(* Logix 5000 project; controller PBS_Perfusion vendor 1 type 14 code 217 rev 32.14; software revision 32.03; part 21 of 27 *)
(* tags used below, declared in another part *)
   ONS : DINT[3];
   REAL : DINT;

ADD_ON_INSTRUCTION P_VSD   (* revision 4.10 .01 Release, vendor Rockwell Automation, ExecutePrescan, ExecuteEnableInFalse *)
// Variable Speed Drive
// Revision note:
// See Instruction Help for a summary of changes, and see 4.10 Release Notes for details.
// Help:
// Copyright © Rockwell Automation, Inc.  All Rights Reserved.
// This Instruction controls and monitors a Variable-Speed (AC or DC) Drive
// and provides:
// *  Starting drive, stopping drive, jogging drive, setting speed reference and setting direction
// *  Monitoring of run feedback, display of actual drive status, including accel, decel, direction, speed
// *  Detection of Failure to Start, Failure to Stop, Drive Fault/Not Ready
// *  Monitoring of Permissive conditions to allow starting
// *  Monitoring of Interlock conditions to stop drive or prevent starting
// *  Simulation, providing feedback of a working drive while disabling outputs
// *  Monitoring of I/O communication faults
// *  Alarms for Fail to Start, Fail to Stop, Interlock Trip, Drive Fault/Not Ready, I/O Fault
// *  Operation in Hand, Maintenance, Override, Program and Operator Modes
// *  "Available" status for use by automation logic to know whether drive
//       can be controlled by other objects.
// *  Horn output for audible alert prior to starting motor.
// Command Sources are arbitrated by a P_CmdSrc Add-On Instruction instance.
// Command Sources: Operator, External, Program, Override, Maintenance, Out of
// Service, Hand.  Alarms are provided by P_Alarm Add-On Instruction instances.
// SUMMARY OF CHANGES FROM PREVIOUS VERSION (4.10.00)
// See 4.10 Release Notes for details.
// * Corrected handling of Start Horn on shed conditions.
// * Modified to lock out jog when jog time expires until jog commands are cleared
// * Modified to handle overlapping Horn and Jog times.
// SUMMARY OF CHANGES FROM PREVIOUS VERSION (4.00.02)
// See 4.10 Release Notes for details.
// * Changed availability to use input availability from interlocks.
// * Added Horn Status, Horn Inhibit.
// * Updated to P_CmdSrc V4.10.00.
// * Modified simulated run feedback to handle run at zero speed ref.
// * Added Cfg_HasMoreObj.
// SUMMARY OF CHANGES FROM PREVIOUS VERSION (4.00.00)
// See 4.00 Release Notes for details.
// * Corrected handling Allow Local when horn is enabled.
// SUMMARY OF CHANGES FROM PREVIOUS VERSION (3.5-11)
// See 4.00 Release Notes for details.
// * Changed "Mode" to "Command Source".
// * Added audible alert on commanded start.  Added unacked alarm count.
// * Changed Inf_ items to HMI_, and added Cfg_Area for security.
// * Changed Start / Stop / Fwd / Rev / Jog to StartFwd / StartRev /Stop / JogFwd / JogRev.
// * Deleted Cfg_PCmdClear; all Program Commands are now self-clearing.
// * All OCmds/MCmds and ORdys/MRdys are now Local Tags.
// * Added Sts_RdyAck and Sts_RdyReset for use by external objects.
// * Aligned ready bit naming with command bit names.
// * Added configurable decimal places for display on HMI.
// * Modifications to Output Datalink clamp limit restrictions / checking.
// * Changed delay / time configuration items to REAL seconds.
// * Updated Val_Sts to common enumeration across all motors and drives.
VAR_IN_OUT
   Ref_FaultCodeList : P_DescList[1]; {required}   // Tag containing List of Fault Codes (DINT) and their Descriptions (STRING)
END_VAR
VAR_INPUT
   Inp_SpeedFdbk : REAL; {visible}   // Speed Feedbak in Drive Units (typ. 0-32767 = 0 to max freq.)
   Inp_LastFaultCode : DINT; {visible}   // Most recent drive fault code (enumeration)
   Inp_Datalink : REAL;   // Auxiliary Signal (datalink) Input in Drive (raw) Units
   Inp_Ready : BOOL := 1; {visible}   // 1=Drive is ready to run
   Inp_Running : BOOL; {visible}   // 1=Drive is Running (active)
   Inp_CommandDir : BOOL := 1; {visible}   // 1=Drive is commanded Forward, 0=Drive is commanded Reverse
   Inp_ActualDir : BOOL := 1; {visible}   // 1=Drive is running Forward, 0=Drive is running Reverse
   Inp_Accelerating : BOOL; {visible}   // 1=Drive is accelerating
   Inp_Decelerating : BOOL; {visible}   // 1=Drive is decelerating
   Inp_Alarm : BOOL; {visible}   // 1=Drive has an Alarm Condition (see drive display or manual)
   Inp_Faulted : BOOL; {visible}   // 1=Drive has Faulted (see drive display or manual)
   Inp_AtSpeed : BOOL; {visible}   // 1=Drive is at commanded speed
   Inp_FwdPermOK : BOOL := 1; {visible}   // 1=Permissives OK, drive can start Forward
   Inp_FwdNBPermOK : BOOL := 1; {visible}   // 1=Non-Bypassable Permissives OK, drive can start Forward
   Inp_RevPermOK : BOOL := 1; {visible}   // 1=Permissives OK, drive can start Reverse
   Inp_RevNBPermOK : BOOL := 1; {visible}   // 1=Non-Bypassable Permissives OK, motor can start Reverse
   Inp_IntlkOK : BOOL := 1; {visible}   // 1=Interlocks OK, drive can start/run
   Inp_NBIntlkOK : BOOL := 1; {visible}   // 1=Non-Bypassable Interlocks OK, drive can start/run
   Inp_IntlkAvail : BOOL;   // 1 = Interlock Availibility OK
   Inp_IOFault : BOOL;   // Input Communication Status 0=OK, 1=fail
   Inp_Sim : BOOL;   // 1=Simulate working drive; 0=Start/Stop/ Monitor actual drive
   Inp_Hand : ALIAS FOR CmdSrc.Inp_Hand;
   Inp_Ovrd : ALIAS FOR CmdSrc.Inp_Ovrd;
   Inp_OvrdCmd : DINT;   // Override Command: 0=None, 1=Stop, 2=Start Fwd 3=Start Rev
   Inp_OvrdSpeed : REAL;   // Value to set Speed Reference in Override Mode (SpeedRef EU)
   Inp_OvrdOutDatalink : REAL;   // Value to set Output Datalink in Override Mode (OutDatalink EU)
   Inp_ExtInh : ALIAS FOR CmdSrc.Inp_ExtInh;
   Inp_HornInh : BOOL;   // 1 = Inhibit audible alert, 0 = Alllow audible alert
   Inp_Reset : BOOL;   // 1=Reset Shed Latches and Cleared Alarms
   Cfg_HasReverse : BOOL;   // 1=Drive can be run reverse, 0=Forward only
   Cfg_HasJog : BOOL;   // 1=Drive Jog Command enabled/visible, 0=Drive Jog Command not allowed
   Cfg_AllowLocal : BOOL;   // 1=Allow Local Start/Stop without alarm, 0=Start/Stop from HMI/prog only
   Cfg_HasRunFdbk : BOOL;   // 1=Drive provides feedback signal on Inp_Running when running
   Cfg_UseRunFdbk : BOOL;   // 1=Drive run feedback should be used for failure checking
   Cfg_HasSpeedFdbk : BOOL;   // 1=Drive provides speed feedback on Inp_SpeedFdbk
   Cfg_UseSpeedFdbk : BOOL := 1;   // 1=Drive speed determines running state, 0=state determined by drive Active input bit
   Cfg_HasInpDatalink : BOOL;   // 1=A signal is connected to Inp_Datalink
   Cfg_HasOutDatalink : BOOL;   // 1=A signal is connected to Out_Datalink
   Cfg_HasFwdPermObj : BOOL;   // 1=Tells HMI a P_Perm is connected to Inp_FwdPerm
   Cfg_HasRevPermObj : BOOL;   // 1=Tells HMI a P_Perm is connected to Inp_RevPerm
   Cfg_HasIntlkObj : BOOL;   // 1=Tells HMI a P_Intlk is connected to Inp_Intlk
   Cfg_HasResInhObj : BOOL;   // 1=Tells HMI a P_ResInh Restart Inhibit is connected
   Cfg_HasRunTimeObj : BOOL;   // 1=Tells HMI a P_RunTime is connected
   Cfg_HasMoreObj : BOOL;   // 1=Tells HMI an object with more info is available
   Cfg_SetTrack : BOOL := 1;   // 1=Settings track for unselected sources, 0=no tracking
   Cfg_SetTrackOvrdHand : BOOL;   // 1=Prog/Oper/Ext Settings track Override/Hand
   Cfg_OperStopPrio : BOOL;   // 1=OCmd_Stop any time, 0=OCmd_Stop only when Oper selected
   Cfg_ExtStopPrio : BOOL;   // 1=XCmd_Stop any time, 0=XCmd_Stop only when Ext selected
   Cfg_OCmdResets : BOOL;   // 1=New drive OCmd resets shed latches and cleared alarms, 0=OCmdReset req'd.
   Cfg_XCmdResets : BOOL;   // 1=New drive XCmd resets shed latches and cleared alarms, 0=XCmdReset req'd.
   Cfg_OvrdPermIntlk : BOOL;   // 1=Override ignores Bypassable Perm/ Intlk; 0=always use Perm/Intlk
   Cfg_ShedOnFailToStart : BOOL := 1;   // 1=Stop Motor and Alarm on Fail to Start; 0=Alarm only on Fail to Start
   Cfg_ShedOnIOFault : BOOL := 1;   // 1=Stop Motor and Alarm on I/O Fault; 0=Alarm only on I/O Fault
   Cfg_SimScaleEU : BOOL;   // 1=In simulation, scale Speed Ref EU to Speed Fdbk EU
   Cfg_SimScaleRaw : BOOL;   // 1=In simulation, scale Speed Ref EU to raw, then raw to Speed Fdbk EU
   Cfg_DecPlcs : DINT := 2;   // Number of decimal places for speed ref/fdbk display (0..6)
   Cfg_InpDLDecPlcs : DINT := 2;   // Number of decimal places for Input Datalink display (0..6)
   Cfg_OutDLDecPlcs : DINT := 2;   // Number of decimal places for Output Datalink display (0..6)
   Cfg_HasFailToStartAlm : ALIAS FOR FailToStart.Cfg_Exists;   // 1=Fail to Start Alarm exists and will be checked
   Cfg_HasFailToStopAlm : ALIAS FOR FailToStop.Cfg_Exists;   // 1=Fail to Stop Alarm exists and will be checked
   Cfg_HasIntlkTripAlm : ALIAS FOR IntlkTrip.Cfg_Exists;   // 1=Interlock Trip Alarm exists and will be checked
   Cfg_HasDriveFaultAlm : ALIAS FOR DriveFault.Cfg_Exists;   // 1=Drive Fault alarm exists and will be checked
   Cfg_HasIOFaultAlm : ALIAS FOR IOFault.Cfg_Exists;   // 1=I/O Fault Alarm exists and will be checked
   Cfg_FailToStartResetReqd : ALIAS FOR FailToStart.Cfg_ResetReqd;   // 1=Reset requied to clear Fail to Start Alarm
   Cfg_FailToStopResetReqd : ALIAS FOR FailToStop.Cfg_ResetReqd;   // 1=Reset required to clear Fail to Stop Alarm
   Cfg_IntlkTripResetReqd : ALIAS FOR IntlkTrip.Cfg_ResetReqd;   // 1=Reset required to clear Interlock Trip Alarm
   Cfg_DriveFaultResetReqd : ALIAS FOR DriveFault.Cfg_ResetReqd;   // 1=Reset required to clear Drive Fault Alarm
   Cfg_IOFaultResetReqd : ALIAS FOR IOFault.Cfg_ResetReqd;   // 1=Reset required to clear I/O Fault Alarm
   Cfg_FailToStartAckReqd : ALIAS FOR FailToStart.Cfg_AckReqd;   // 1=Acknowledge required for Fail to Start Alarm
   Cfg_FailToStopAckReqd : ALIAS FOR FailToStop.Cfg_AckReqd;   // 1=Acknowledge required for Fail to Stop Alarm
   Cfg_IntlkTripAckReqd : ALIAS FOR IntlkTrip.Cfg_AckReqd;   // 1=Acknowledge required for Interlock Trip Alarm
   Cfg_DriveFaultAckReqd : ALIAS FOR DriveFault.Cfg_AckReqd;   // 1=Acknowledge required for Drive Fault Alarm
   Cfg_IOFaultAckReqd : ALIAS FOR IOFault.Cfg_AckReqd;   // 1=Acknowledge required for I/O Fault Alarm
   Cfg_FailToStartSeverity : ALIAS FOR FailToStart.Cfg_Severity;   // Fail To Start Alarm Severity: 1..250=Low, 251..500=Medium, 501..750=High, 751..1000=Urgent
   Cfg_FailToStopSeverity : ALIAS FOR FailToStop.Cfg_Severity;   // Fail To Stop Alarm Severity: 1..250=Low, 251..500=Medium, 501..750=High, 751..1000=Urgent
   Cfg_IntlkTripSeverity : ALIAS FOR IntlkTrip.Cfg_Severity;   // Interlock Trip Alarm Severity: 1..250=Low, 251..500=Medium, 501..750=High, 751..1000=Urgent
   Cfg_DriveFaultSeverity : ALIAS FOR DriveFault.Cfg_Severity;   // Drive Fault Alarm Severity: 1..250=Low, 251..500=Medium, 501..750=High, 751..1000=Urgent
   Cfg_IOFaultSeverity : ALIAS FOR IOFault.Cfg_Severity;   // I/O Fault Alarm Severity: 1..250=Low, 251..500=Medium, 501..750=High, 751..1000=Urgent
   Cfg_MinSpdRef : REAL;   // Minimum Speed Reference in EU (for limiting)
   Cfg_MaxSpdRef : REAL := 60.0;   // Maximum Speed Reference in EU (for limiting)
   Cfg_SpeedRefRawMin : REAL;   // Speed Reference Minimum in Drive (raw) Units (for scaling)
   Cfg_SpeedRefRawMax : REAL := 32767.0;   // Speed Reference Maximum in Drive (raw) Units (for scaling)
   Cfg_SpeedRefEUMin : REAL;   // Speed Reference Minimum in Engineering Units (for scaling)
   Cfg_SpeedRefEUMax : REAL := 130.0;   // Speed Reference Maximum in Engineering Units (for scaling)
   Cfg_SpeedFdbkRawMin : REAL;   // Speed Feedback Minimum in Drive (raw) Units (for scaling)
   Cfg_SpeedFdbkRawMax : REAL := 32767.0;   // Speed Feedback Maximum in Drive (raw) Units (for scaling)
   Cfg_SpeedFdbkEUMin : REAL;   // Speed Feedback Minimum in Engineering Units (for scaling)
   Cfg_SpeedFdbkEUMax : REAL := 130.0;   // Speed Feedback Maximum in Engineering Units (for scaling)
   Cfg_InpDatalinkRawMin : REAL;   // Input Datalink Minimum in Drive (raw) Units (for scaling)
   Cfg_InpDatalinkRawMax : REAL := 4095.0;   // Input Datalink Maximum in Drive (raw) Units (for scaling)
   Cfg_InpDatalinkEUMin : REAL;   // Input Datalink Minimum in Engineering Units (for scaling)
   Cfg_InpDatalinkEUMax : REAL := 409.5;   // Input Datalink Maximum in Engineering Units (for scaling)
   Cfg_OutDatalinkMin : REAL;   // Minimum Output Datalink in EU (for limiting)
   Cfg_OutDatalinkMax : REAL := 100.0;   // Maximum Output Datalink in EU (for limiting)
   Cfg_OutDatalinkRawMin : REAL;   // Output Datalink Minimum in Drive (raw) Units (for scaling)
   Cfg_OutDatalinkRawMax : REAL := 4095.0;   // Output Datalink Maximum in Drive (raw) Units (for scaling)
   Cfg_OutDatalinkEUMin : REAL;   // Output Datalink Minimum in Engineering Units (for scaling)
   Cfg_OutDatalinkEUMax : REAL := 409.5;   // Output Datalink Maximum in Engineering Units (for scaling)
   Cfg_StartHornT : REAL;   // Time to sound audible on commanded start (sec) (0=disabled)
   Cfg_SimRampT : REAL := 10.0;   // Time to ramp speed fdbk when in Simulation (sec)
   Cfg_FailToStartT : REAL := 15.0;   // Time after Start to get Run Feedback before Fault (sec)
   Cfg_FailToStopT : REAL := 15.0;   // Time after Stop to drop Run Feedback before Fault (sec)
   Cfg_ResetPulseT : REAL := 2.0;   // Time to pulse Out_Reset to clear drive fault
   Cfg_MaxJogT : REAL;   // Maximum jog time (sec, 0=unlimited)
   Cfg_OperKeep : SINT;   // Oper keeps control in Prog / Ext: .0=Reference, .1=Start/Stop/Fwd/ Rev, .3=OutDatalink
   Cfg_ProgKeep : SINT;   // Prog keeps control in Oper / Ext: .0=Reference, .1=Start/Stop/Fwd/ Rev, .3=OutDatalink
   Cfg_ExtKeep : SINT;   // Ext keeps control in Prog / Oper: .0=Reference, .1=Start/Stop/Fwd/ Rev, .3=OutDatalink
   PSet_SpeedRef : REAL;   // Program Setting of Speed Reference (EU)
   PSet_OutDatalink : REAL;   // Program Setting of Output Datalink (EU)
   PSet_Owner : DINT;   // Program Owner Request ID (non-zero) or Release (zero)
   XSet_SpeedRef : REAL;   // External Setting of Speed Reference (EU)
   XSet_OutDatalink : REAL;   // External Setting of Output Datalink (EU)
   PCmd_StartFwd : BOOL;   // Program Command to Start Drive Forward
   PCmd_StartRev : BOOL;   // Program Command to Start Drive Reverse
   PCmd_Stop : BOOL;   // Program Command to Stop Drive
   PCmd_Prog : ALIAS FOR CmdSrc.PCmd_Prog;
   PCmd_Oper : ALIAS FOR CmdSrc.PCmd_Oper;
   PCmd_Lock : ALIAS FOR CmdSrc.PCmd_Lock;
   PCmd_Unlock : ALIAS FOR CmdSrc.PCmd_Unlock;
   PCmd_Normal : ALIAS FOR CmdSrc.PCmd_Normal;
   PCmd_Reset : BOOL;   // Program Command to Reset drive fault and all Alarms requiring Reset
   PCmd_FailToStartAck : ALIAS FOR FailToStart.PCmd_Ack;   // Program Command to Acknowledge Fail to Start Alarm
   PCmd_FailToStartSuppress : ALIAS FOR FailToStart.PCmd_Suppress;   // Program Command to Suppress Fail to Start Alarm
   PCmd_FailToStartUnsuppress : ALIAS FOR FailToStart.PCmd_Unsuppress;   // Program Command to Unsuppress Fail to Start Alarm
   PCmd_FailToStartUnshelve : ALIAS FOR FailToStart.PCmd_Unshelve;   // Program Command to Unshelve Fail to Start Alarm
   PCmd_FailToStopAck : ALIAS FOR FailToStop.PCmd_Ack;   // Program Command to Acknowledge Fail to Stop Alarm
   PCmd_FailToStopSuppress : ALIAS FOR FailToStop.PCmd_Suppress;   // Program Command to Suppress Fail to Stop Alarm
   PCmd_FailToStopUnsuppress : ALIAS FOR FailToStop.PCmd_Unsuppress;   // Program Command to Unsuppress Fail to Stop Alarm
   PCmd_FailToStopUnshelve : ALIAS FOR FailToStop.PCmd_Unshelve;   // Program Command to Unshelve Fail to Stop Alarm
   PCmd_IntlkTripAck : ALIAS FOR IntlkTrip.PCmd_Ack;   // Program Command to Acknowledge Interlock Trip Alarm
   PCmd_IntlkTripSuppress : ALIAS FOR IntlkTrip.PCmd_Suppress;   // Program Command to Suppress Interlock Trip Alarm
   PCmd_IntlkTripUnsuppress : ALIAS FOR IntlkTrip.PCmd_Unsuppress;   // Program Command to Unsuppress Interlock Trip Alarm
   PCmd_IntlkTripUnshelve : ALIAS FOR IntlkTrip.PCmd_Unshelve;   // Program Command to Unshelve Interlock Trip Alarm
   PCmd_DriveFaultAck : ALIAS FOR DriveFault.PCmd_Ack;   // Program Command to Acknowledge Drive Fault Alarm
   PCmd_DriveFaultSuppress : ALIAS FOR DriveFault.PCmd_Suppress;   // Program Command to Suppress Drive Fault Alarm
   PCmd_DriveFaultUnsuppress : ALIAS FOR DriveFault.PCmd_Unsuppress;   // Program Command to Unsuppress Drive Fault Alarm
   PCmd_DriveFaultUnshelve : ALIAS FOR DriveFault.PCmd_Unshelve;   // Program Command to Unshelve Drive Fault Alarm
   PCmd_IOFaultAck : ALIAS FOR IOFault.PCmd_Ack;   // Program Command to Acknowledge I/O Fault Alarm
   PCmd_IOFaultSuppress : ALIAS FOR IOFault.PCmd_Suppress;   // Program Command to Suppress I/O Fault Alarm
   PCmd_IOFaultUnsuppress : ALIAS FOR IOFault.PCmd_Unsuppress;   // Program Command to Unsuppress I/O Fault Alarm
   PCmd_IOFaultUnshelve : ALIAS FOR IOFault.PCmd_Unshelve;   // Program Command to Unshelve I/O Fault Alarm
   MCmd_Rel : ALIAS FOR CmdSrc.MCmd_Rel;
   OCmd_Unlock : ALIAS FOR CmdSrc.OCmd_Unlock;
   XCmd_StartFwd : BOOL;   // External Command to Start Drive Forward
   XCmd_StartRev : BOOL;   // External Command to Start Drive Reverse
   XCmd_Stop : BOOL;   // External Command to Stop Drive
   XCmd_JogFwd : BOOL;   // External Command to Jog Drive Forward
   XCmd_JogRev : BOOL;   // External Command to Jog Drive Reverse
   XCmd_Acq : ALIAS FOR CmdSrc.XCmd_Acq;
   XCmd_Rel : ALIAS FOR CmdSrc.XCmd_Rel;
   XCmd_Reset : BOOL;   // Ext Cmd to clear shed latches and cleared alarms
END_VAR
VAR_OUTPUT
   Out_SpeedRef : REAL; {access Read Only, visible}   // Drive Speed Reference in Drive Units (typ. 0-32767 = 0 to max freq.)
   Out_Datalink : REAL; {access Read Only, visible}   // Auxiliary Signal (datalink) Output in Drive (raw) Units
   Out_Run : BOOL; {access Read Only}   // 1=Start/Run Drive, 0=Stop Drive (for held starter type)
   Out_Stop : BOOL; {access Read Only, visible}   // 1=Stop Drive, 0=drive left in current state
   Out_Start : BOOL; {access Read Only, visible}   // 1=Start Drive, 0=drive left in current state
   Out_Jog : BOOL; {access Read Only, visible}   // 1=Jog drive at Jog Speed, -->0=stop jogging
   Out_ClearFault : BOOL; {access Read Only, visible}   // 1=Attempt to clear Drive Fault
   Out_Fwd : BOOL; {access Read Only, visible}   // 1=Set drive direction to Forward
   Out_Rev : BOOL; {access Read Only, visible}   // 1=Set drive direction to Reverse
   Out_Horn : BOOL; {access Read Only, visible}   // 1=Sound audible prior to commanded motor start
   Val_SpeedRef : REAL; {access Read Only, visible}   // Speed Reference (target) to drive
   Val_SpeedFdbk : REAL; {access Read Only, visible}   // Speed Feedback (actual) from drive
   Val_InpDatalink : REAL; {access Read Only, visible}   // Input Datalink value from drive
   Val_OutDatalink : REAL; {access Read Only, visible}   // Output Datalink value to drive
   Val_SpeedRefEUMin : REAL; {access Read Only}   // Minimum of Speed Reference = MIN (Cfg_SpeedFdbkEUMin, Cfg_SpeedFdbkEUMax)
   Val_SpeedRefEUMax : REAL := 130.0; {access Read Only}   // Maximum of Speed Reference = MAX (Cfg_SpeedFdbkEUMin, Cfg_SpeedFdbkEUMax)
   Val_SpeedFdbkEUMin : REAL; {access Read Only}   // Minimum of Speed Feedback = MIN (Cfg_SpeedFdbkEUMin, Cfg_SpeedFdbkEUMax)
   Val_SpeedFdbkEUMax : REAL := 130.0; {access Read Only}   // Maximum of Speed Feedback = MAX (Cfg_SpeedFdbkEUMin, Cfg_SpeedFdbkEUMax)
   Val_LastFaultCode : DINT; {access Read Only}   // Most recent drive fault code (enumeration)
   SrcQ_IO : DINT; {access Read Only}   // Source and Quality of primary I/O (enumeration)
   SrcQ : DINT; {access Read Only}   // Source and Quality of primary Val/Sts (enumeration)
   Val_Cmd : DINT; {access Read Only}   // Device Command 0=None, 1=Stop, 2=StartFwd 3=StartRev 4=JogFwd 5=JogRev
   Val_Fdbk : DINT; {access Read Only}   // Device Feedback 0=Stopped, 1=Running Fwd 2=Running Rev 3=Accelerating 4=Decelerating
   Val_Sts : DINT; {access Read Only}   // Device Sts: 0=? 1=Stopped 2=RunFwd 3=RunRev 4=RunSlow 5=StartFwd 6=StartRev 7=StartSlow 8=JogFwd 9=JogRev 10=Stopping
   Val_Fault : DINT; {access Read Only, visible}   // Device Fault Status 0=None, 16=Fail to Start, 17 = Fail to Stop, 18=Drive Fault, 32=I/O Fault, 34=Config Error
   Val_NotifyAll : DINT; {access Read Only}   // Highest Alarm prio and ack status this object + channel (enum)
   Val_UnackAlmC : DINT; {access Read Only}   // Count of Unacknowledged Alarms
   Val_Owner : DINT; {access Read Only}   // Current Object Owner ID (0=not owned)
   Sts_Stopped : BOOL; {access Read Only, visible}   // 1=Drive requested to stop and is confirmed stopped
   Sts_StartingFwd : BOOL; {access Read Only, visible}   // 1=Drive requested to run forward and awaiting run feedback
   Sts_StartingRev : BOOL; {access Read Only, visible}   // 1=Drive requested to run reverse and awaiting run feedback
   Sts_RunningFwd : BOOL; {access Read Only, visible}   // 1=Drive requested to run and is confirmed running forward
   Sts_RunningRev : BOOL; {access Read Only, visible}   // 1=Drive requested to run and is confirmed running reverse
   Sts_StoppingFwd : BOOL; {access Read Only, visible}   // 1=Drive running forward requested to stop and awaiting stopped feedback
   Sts_StoppingRev : BOOL; {access Read Only, visible}   // 1=Drive running reverse requested to stop and awaiting stopped feedback
   Sts_JoggingFwd : BOOL; {access Read Only, visible}   // 1=Drive requested to Jog Forward
   Sts_JoggingRev : BOOL; {access Read Only, visible}   // 1=Drive requested to Jog Reverse
   Sts_Horn : BOOL; {access Read Only}   // 1=Motor Horn Active
   Sts_CommandDir : BOOL; {access Read Only}   // 1=Drive commanded to Forward, 0=Reverse
   Sts_ActualDir : BOOL; {access Read Only, visible}   // 1=Drive Actual direction is Forward, 0=Reverse
   Sts_Accel : BOOL; {access Read Only}   // 1=Drive is Accelerating
   Sts_Decel : BOOL; {access Read Only}   // 1=Drive is Decelerating
   Sts_NotReady : BOOL; {access Read Only}   // 1=Drive is Not Ready (cannot be started) Check alarms, stops, faults
   Sts_Alarm : BOOL; {access Read Only, visible}   // 1=Drive has an Alarm (see drive display or manual)
   Sts_AtSpeed : BOOL; {access Read Only, visible}   // 1=Drive is running at reference speed
   Sts_SpeedLimited : BOOL; {access Read Only, visible}   // 1=Speed Reference Setting exceeds configured Max/Min limit
   Sts_Available : BOOL; {access Read Only, visible}   // 1=Drive available for control by automation (Prog)
   Sts_Bypass : BOOL; {access Read Only}   // 1=Bypassable Interlocks and Permissives are Bypassed
   Sts_BypActive : BOOL; {access Read Only}   // 1=Bypassing Active (Bypassed or Maintenance)
   Sts_NotRdy : BOOL; {access Read Only}   // 1=Device Not Ready, see detail bits for reason
   Nrdy_CfgErr : BOOL; {access Read Only}   // 1=Device Not Ready: Configuration Error
   Nrdy_DriveNR : BOOL; {access Read Only}   // 1=Device Note Ready: Drive Not Ready
   Nrdy_Fail : BOOL; {access Read Only}   // 1=Device Not Ready: Device Failure (Shed Requires Reset)
   Nrdy_Intlk : BOOL; {access Read Only, visible}   // 1=Device Not Ready: Interlock Not OK
   Nrdy_IOFault : BOOL; {access Read Only}   // 1=Device Not Ready: I/O Fault (Shed Requires Reset)
   Nrdy_OoS : BOOL; {access Read Only}   // 1=Device Not Ready: Device is Out of Service
   Nrdy_Perm : BOOL; {access Read Only}   // 1=Device Not Ready: Permissive Not OK
   Nrdy_PrioStop : BOOL; {access Read Only}   // 1=Device Not Ready: Oper/Ext Priority Stop Requires Reset
   Nrdy_Trip : BOOL; {access Read Only}   // 1=Device not Ready: Deivce Tripped (Drive Fault)
   Sts_MaintByp : BOOL; {access Read Only}   // 1=A Maintenance Bypass is Active, display icon
   Sts_AlmInh : BOOL; {access Read Only}   // 1=An Alarm is Shelved, Disabled or Suppressed, display icon
   Sts_Err : BOOL; {access Read Only, visible}   // 1=Error in Config: see detail bits for reason
   Err_Timer : BOOL; {access Read Only}   // 1=Error in Config: Invalid Check or Reset Pulse Time (use 0 to 2147483)
   Err_Sim : BOOL; {access Read Only}   // 1=Error in Config: simulation timer preset: use 0 to 2147483)
   Err_Alarm : BOOL; {access Read Only}   // 1=Error in Config: Alarm Min On Time, Shelf Time, Severity
   Err_FdbkRaw : BOOL; {access Read Only}   // 1=Erron in Config: Speed Fdbk Raw Min = Max
   Err_FdbkEU : BOOL; {access Read Only}   // 1=Error in Config: Speed Fdbk EU Min = Max
   Err_RefLim : BOOL; {access Read Only}   // 1=Error in Config: Speed Ref Limit Min > Max
   Err_RefEU : BOOL; {access Read Only}   // 1=Error in Config: Speed Ref EU Min = Max
   Err_RefRaw : BOOL; {access Read Only}   // 1=Error in Config: Speed Ref Raw Min = Max
   Err_InpDLRaw : BOOL; {access Read Only}   // 1=Error in Config: Input Datalink Raw Min = Max
   Err_InpDLEU : BOOL; {access Read Only}   // 1=Error in Config: Input Datalink EU Min = Max
   Err_OutDLLim : BOOL; {access Read Only}   // 1=Error in Config: Output Datalink Limits Min > Max
   Err_OutDLEU : BOOL; {access Read Only}   // 1=Error in Config: Output Datalink EU Min = Max
   Err_OutDLRaw : BOOL; {access Read Only}   // 1=Error in Config: Output Datalink Raw Min = Max
   Sts_Hand : ALIAS FOR CmdSrc.Sts_Hand; {access Read Only, visible}
   Sts_OoS : ALIAS FOR CmdSrc.Sts_OoS; {access Read Only, visible}
   Sts_Maint : ALIAS FOR CmdSrc.Sts_Maint; {access Read Only, visible}
   Sts_Ovrd : ALIAS FOR CmdSrc.Sts_Ovrd; {access Read Only, visible}
   Sts_Ext : ALIAS FOR CmdSrc.Sts_Ext; {access Read Only, visible}
   Sts_Prog : ALIAS FOR CmdSrc.Sts_Prog; {access Read Only, visible}
   Sts_ProgLocked : ALIAS FOR CmdSrc.Sts_ProgLocked; {access Read Only}
   Sts_Oper : ALIAS FOR CmdSrc.Sts_Oper; {access Read Only, visible}
   Sts_OperLocked : ALIAS FOR CmdSrc.Sts_OperLocked; {access Read Only}
   Sts_Normal : ALIAS FOR CmdSrc.Sts_Normal; {access Read Only}
   Sts_ExtReqInh : ALIAS FOR CmdSrc.Sts_ExtReqInh; {access Read Only}
   Sts_ProgReqInh : ALIAS FOR CmdSrc.Sts_ProgReqInh; {access Read Only}
   Sts_MAcqRcvd : ALIAS FOR CmdSrc.Sts_MAcqRcvd; {access Read Only}
   Sts_RdyReset : ALIAS FOR ORdy_Reset; {access Read Only}   // 1=A latched alarm or shed condition is ready to be reset
   Sts_RdyAck : BOOL; {access Read Only}   // 1=An alarm is ready to be acknowledged
   Sts_FailToStart : ALIAS FOR FailToStart.Inp;   // 1=Drive Failed to Start (One-Shot)
   Alm_FailToStart : ALIAS FOR FailToStart.Alm;   // 1=Drive Fail to Start Alarm
   Ack_FailToStart : ALIAS FOR FailToStart.Ack;   // 1=Fail to Start Alarm has been acknowledged
   Sts_FailToStartDisabled : ALIAS FOR FailToStart.Disabled;   // 1=Fail to Start Alarm has been Disabled by Maintenance
   Sts_FailToStartShelved : ALIAS FOR FailToStart.Shelved;   // 1=Fail to Start Alarm has been Shelved by Operator
   Sts_FailToStartSuppressed : ALIAS FOR FailToStart.Suppressed;   // 1=Fail to Start Alarm has been Suppressed by Program
   Sts_FailToStop : ALIAS FOR FailToStop.Inp;   // 1=Drive Failed to Stop
   Alm_FailToStop : ALIAS FOR FailToStop.Alm;   // 1=Drive Fail to Stop Alarm
   Ack_FailToStop : ALIAS FOR FailToStop.Ack;   // 1=Fail to Stop Alarm has been acknowledged
   Sts_FailToStopDisabled : ALIAS FOR FailToStop.Disabled;   // 1=Fail to Stop Alarm has been Disabled by Maintenance
   Sts_FailToStopShelved : ALIAS FOR FailToStop.Shelved;   // 1=Fail to Stop Alarm has been Shelved by Operator
   Sts_FailToStopSuppressed : ALIAS FOR FailToStop.Suppressed;   // 1=Fail to Stop Alarm has been Suppressed by Program
   Sts_IntlkTrip : ALIAS FOR IntlkTrip.Inp;   // 1=Drive was stopped by an Interlock NOT OK (One-Shot)
   Alm_IntlkTrip : ALIAS FOR IntlkTrip.Alm;   // 1=Alarm: Drive stopped by an Interlock NOT OK
   Ack_IntlkTrip : ALIAS FOR IntlkTrip.Ack;   // 1=Interlock Trip Alarm has been acknowledged
   Sts_IntlkTripDisabled : ALIAS FOR IntlkTrip.Disabled;   // 1=Interlock Trip Alarm has been Disabled by Maintenance
   Sts_IntlkTripShelved : ALIAS FOR IntlkTrip.Shelved;   // 1=Interlock Trip Alarm has been Shelved by Operator
   Sts_IntlkTripSuppressed : ALIAS FOR IntlkTrip.Suppressed;   // 1=Interlock Trip Alarm has been Suppressed by Program
   Sts_DriveFault : ALIAS FOR DriveFault.Inp;   // 1=Drive Fault (see drive display or manual)
   Alm_DriveFault : ALIAS FOR DriveFault.Alm;   // 1=Alarm: Drive Fault (see drive display or manual)
   Ack_DriveFault : ALIAS FOR DriveFault.Ack;   // 1=Drive Fault Alarm has been acknowledged
   Sts_DriveFaultDisabled : ALIAS FOR DriveFault.Disabled;   // 1=Drive Fault Alarm has been Disabled by Maintenance
   Sts_DriveFaultShelved : ALIAS FOR DriveFault.Shelved;   // 1=Drive Fault Alarm has been Shelved by Operator
   Sts_DriveFaultSuppressed : ALIAS FOR DriveFault.Suppressed;   // 1=Drive Fault Alarm has been Suppressed by Program
   Sts_IOFault : ALIAS FOR IOFault.Inp;   // I/O Comm Fault Status (0=OK, 1=Bad)
   Alm_IOFault : ALIAS FOR IOFault.Alm;   // 1=I/O Fault Alarm
   Ack_IOFault : ALIAS FOR IOFault.Ack;   // 1=I/O Fault Alarm has been acknowledged
   Sts_IOFaultDisabled : ALIAS FOR IOFault.Disabled;   // 1=I/O Fault Alarm has been Disabled by Maintenance
   Sts_IOFaultShelved : ALIAS FOR IOFault.Shelved;   // 1=I/O Fault Alarm has been Shelved by Operator
   Sts_IOFaultSuppressed : ALIAS FOR IOFault.Suppressed;   // 1=I/O Fault Alarm has been Suppressed by Program
   MRdy_Rel : ALIAS FOR CmdSrc.MRdy_Rel; {access Read Only}
   ORdy_Unlock : ALIAS FOR CmdSrc.ORdy_Unlock; {access Read Only}
   P_VSD : BOOL;   // Unique Parameter Name for auto - discovery
END_VAR
VAR
   CmdSrc : P_CmdSrc := (Cfg_HasOper := 1, Cfg_HasOperLocked := 1, Cfg_HasProg := 1, Cfg_HasProgLocked := 1, Cfg_HasMaint := 1, Cfg_HasMOoS := 1, Cfg_OvrdOverLock := 1, Sts_bSrc := 1);   // Drive Mode Selection
   IOFault : P_Alarm := (Cfg_AckReqd := 1, Cfg_AllowShelve := 1, Cfg_AllowDisable := 1, Cfg_Severity := 1000, Cfg_AlmMinOnT := 5, PCfg_AllowExist := 1, Ack := 1);   // I/O Fault Alarm
   IntlkTrip : P_Alarm := (Cfg_AckReqd := 1, Cfg_AllowShelve := 1, Cfg_AllowDisable := 1, Cfg_Severity := 500, Cfg_AlmMinOnT := 5, PCfg_AllowExist := 1, Ack := 1);   // Interlock Trip Alarm
   FailToStop : P_Alarm := (Cfg_AckReqd := 1, Cfg_AllowShelve := 1, Cfg_AllowDisable := 1, Cfg_Severity := 1000, Cfg_AlmMinOnT := 5, PCfg_AllowExist := 1, Ack := 1);   // Drive Failed to Stop Alarm
   FailToStart : P_Alarm := (Cfg_AckReqd := 1, Cfg_AllowShelve := 1, Cfg_AllowDisable := 1, Cfg_Severity := 1000, Cfg_AlmMinOnT := 5, PCfg_AllowExist := 1, Ack := 1);   // Drive Failed to Start Alarm
   Cfg_Tag : STRING_20 := 'P_VSD';   // Tagname for display on HMI
   Cfg_Label : STRING_20 := 'Motor Speed Control';   // Label for graphic symbol displayed on HMI
   Cfg_Desc : STRING_40 := 'Variable Speed Drive';   // Description for display on HMI
   Wrk_Run : BOOL; {access None}   // 1=Drive should be "running", 0=should be "stopped"
   Wrk_StartRetrigT : TIMER; {access None}   // Time to pulse start output on start command retrigger (Maint)
   Wrk_StopRetrigT : TIMER; {access None}   // Time to pulse stop output on stop command retrigger (Maint)
   Wrk_RunFdbk : BOOL; {access None}   // Run Feedback based on mode, simulation, etc. 1=running
   Wrk_Notify : DINT; {access None}   // Buffer for building Val_Notify
   Wrk_Bypass : BOOL; {access None}   // Internal Bypassable Permissives and Interlocks are Bypassed flag
   DriveFault : P_Alarm := (Cfg_AckReqd := 1, Cfg_AllowShelve := 1, Cfg_AllowDisable := 1, Cfg_Severity := 1000, Cfg_AlmMinOnT := 5, PCfg_AllowExist := 1, Ack := 1);   // Drive Faulted Alarm
   Cfg_SpeedRefEU : STRING_8 := 'Hz';   // Speed Reference Engineering Units for display on HMI
   Wrk_SpeedRef : REAL; {access None}   // Working copy of Speed Reference (for limiting)
   Wrk_Rev : BOOL; {access None}   // Working (internal) Direction 1=Reverse 0=Forward (default)
   Wrk_Jog : BOOL; {access None}   // 1=Jog Drive, 0=Drive not jogging
   Wrk_ResetT : TIMER; {access None}   // Reset Output Pulse Timer
   Wrk_ResetONS : BOOL; {access None}   // One-Shot to fire Reset Timer to ensure min. output ON time.
   Cfg_SpeedFdbkEU : STRING_8 := 'Hz';   // Speed Feedback Engineering Units for display on HMI
   Cfg_OutDatalinkLabel : STRING_20;   // Datalink Output Label displayed on faceplate
   Cfg_InpDatalinkLabel : STRING_20;   // Datalink Input Label displayed on faceplate
   Cfg_OutDatalinkEU : STRING_8;   // Datalink Output Engineering Units for display on HMI
   Cfg_InpDatalinkEU : STRING_8;   // Datalink Input Engineering Units for display on HMI
   Wrk_OutDatalink : REAL; {access None}   // Selected Output Datalink setting
   Cfg_RevText : STRING_16 := 'Reverse';   // Name for Reverse Direction, e.g., "Down", "Reverse"
   Cfg_FwdText : STRING_16 := 'Forward';   // Name for Forward Direction, e.g., "Up", "Forward"
   Wrk_StopT : TIMER; {access Read Only}   // Stop Check Timer (for Fail to Stop)
   Wrk_StartT : TIMER; {access Read Only}   // Start Check Timer (for Fail to Start)
   HMI_Tab : SINT;   // Tab to display (FTView ME)
   Wrk_Cmd : DINT; {access None}   // Buffer for building Val_Cmd
   Wrk_Sts : DINT; {access None}   // Buffer for building Val_Sts
   Wrk_Fault : DINT; {access None}   // Buffer for building Val_Fault
   Wrk_Retrigger : BOOL; {access None}   // Maint Start issued while running or Stop while stopped
   Wrk_Step : REAL; {access None}   // Amount to change simulated Speed Fdbk this scan (ramp)
   Wrk_ScanTime : REAL; {access None}   // Seconds since previous scan
   Wrk_ScanT : TIMER := (PRE := 2147483647); {access None}   // Scan Timer (milliseconds, always runs)
   Wrk_SimFdbkTgt : REAL; {access None}   // Speed Ref converted to Speed Fdbk units for simulation: target speed fdbk
   HMI_Type : STRING_16 := 'P_VSD'; {access Read Only}   // Type identifier for HMI navigation
   Wrk_JogT : TIMER; {access Read Only}   // Jog Timer
   Wrk_FaultDescFSC : CONTROL := (LEN := 1); {access None}   // FSC control for Fault Code List search
   Val_FaultDesc : STRING_40; {access Read Only}   // Description of Drive Fault (given LastFaultCode)
   Wrk_OperKeep3ONS : BOOL; {access None}   // Oper Keep bit 3 one-shot store
   Wrk_OperKeep1ONS : BOOL; {access None}   // Oper Keep bit 1 one-shot store
   Wrk_OperKeep0ONS : BOOL; {access None}   // Oper Keep bit 0 one-shot store
   Wrk_ProgKeep3ONS : BOOL; {access None}   // Prog Keep bit 3 one-shot store
   Wrk_ProgKeep1ONS : BOOL; {access None}   // Prog Keep bit 1 one-shot store
   Wrk_ProgKeep0ONS : BOOL; {access None}   // Prog Keep bit 0 one-shot store
   HMI_Lib : STRING_12 := 'RA-BAS'; {access Read Only}   // Display Library for Faceplate call-up
   Wrk_SimScaleEUONS : BOOL; {access None}   // Cfg_SimScaleEU became true this scan
   Wrk_SimScaleRawONS : BOOL; {access None}   // Cfg_SimScaleRaw became true this scan
   Wrk_SrcQ : DINT; {access None}   // Register for building Source / Quality enumeration
   Val_Notify : DINT; {access Read Only}   // Current Alarm Level and Acknowledgement (enumeration)
   Wrk_NotRdyONS : BOOL; {access None}   // Assert Stop on One-Shot of Sts_NotRdy
   Wrk_NotRdy : BOOL; {access None}   // Device Not Ready conditions excluding shed latches
   Wrk_StartInhT : TIMER; {access None}   // Local Start Inhibit Timer
   Wrk_StopInhT : TIMER; {access None}   // Local Stop Inhibit Timer
   Wrk_NoLongerSim : BOOL; {access None}   // Switched from Simulated to Real Drive this scan
   Wrk_Hand : BOOL; {access None}   // Perform Hand Mode alignment with actual device state
   Cfg_Area : STRING_Area := 'area01';   // Process Area for security
   Wrk_UnackAlmC : DINT; {access None}   // Buffer for building Val_UnackAlmC
   Wrk_StartHornT : TIMER; {access None}   // Timer for audible alert or start
   Wrk_StartHorn : BOOL; {access None}   // 1=Sound audible prior to commanded motor start
   Wrk_RevPermOK : BOOL; {access None}   // Reverse Permissives and NB Permissive OK
   Wrk_FwdPermOK : BOOL; {access None}   // Forward Permissives and NB Permissive OK
   OCmd_ResetAckAll : BOOL;   // Oper Cmd to reset shed latches and cleared alarms, plus Acknowledge alarms
   OCmd_Reset : BOOL;   // Oper Cmd to clear shed latches and cleared alarms
   OCmd_JogRev : BOOL;   // Operator Command to Jog Drive Reverse (not cleared by instruction!)
   OCmd_JogFwd : BOOL;   // Operator Command to Jog Drive Forward (not cleared by instruction!)
   OCmd_Stop : BOOL;   // Operator Command to Stop Drive
   OCmd_StartRev : BOOL;   // Operator Command to Start Drive Reverse
   OCmd_StartFwd : BOOL;   // Operator Command to Start Drive Forward
   MCmd_Check : BOOL;   // Maintenance Command to Check (not bypass) all Interlocks and Permissives
   MCmd_Bypass : BOOL;   // Maintenance Command to Bypass all Bypassable Interlocks and Permissives
   OSet_OutDatalink : REAL;   // Operator Setting of Output Datalink (EU)
   OSet_SpeedRef : REAL;   // Operator Setting of Speed Reference (EU)
   ORdy_ResetAckAll : BOOL; {access Read Only}   // 1=Ready for OCmd_ResetAckAll (enables HMI button)
   ORdy_Reset : BOOL; {access Read Only}   // 1=Ready for OCmd_Reset (enables HMI button)
   ORdy_JogRev : BOOL; {access Read Only}   // 1=Ready for OCmd_JogRev (enabled HMI button)
   ORdy_JogFwd : BOOL; {access Read Only}   // 1=Ready for OCmd_JogFwd (enables HMI button)
   ORdy_Stop : BOOL; {access Read Only}   // 1=Ready for OCmd_Stop (enables HMI button)
   ORdy_StartRev : BOOL; {access Read Only}   // 1=Ready for OCmd_StartRev (enables HMI button)
   ORdy_StartFwd : BOOL; {access Read Only}   // 1=Ready for OCmd_StartFwd (enables HMI button)
   ORdy_OSet : BOOL; {access Read Only}   // 1=Ready for OSets (other than Speed Ref) (enables data entry fields)
   ORdy_SpeedRef : BOOL; {access Read Only}   // 1=Ready for OSet_SpeedRef (enables data entry field)
   MRdy_Check : BOOL; {access Read Only}   // 1=Ready for MCmd_Check (enables HMI button)
   MRdy_Bypass : BOOL; {access Read Only}   // 1=Ready for MCmd_Bypass (enables HMI button)
   Wrk_ExtKeep3ONS : BOOL; {access None}   // Ext Keep bit 3 one-shot store
   Wrk_ExtKeep1ONS : BOOL; {access None}   // Ext Keep bit 1 one-shot store
   Wrk_ExtKeep0ONS : BOOL; {access None}   // Ext Keep bit 0 one-shot store
   Wrk_ExtHas3 : BOOL; {access None}   // External has Output Datalink
   Wrk_ExtHas1 : BOOL; {access None}   // External has Commands
   Wrk_ExtHas0 : BOOL; {access None}   // External has Speed Reference
   Wrk_ProgHas3 : BOOL; {access None}   // Program has Output Datalink
   Wrk_ProgHas1 : BOOL; {access None}   // Program has Commands
   Wrk_ProgHas0 : BOOL; {access None}   // Program has Speed Reference
   Wrk_OperHas3 : BOOL; {access None}   // Operator has Output Datalink
   Wrk_OperHas1 : BOOL; {access None}   // Operator has Commands
   Wrk_OperHas0 : BOOL; {access None}   // Operator has Speed Reference
END_VAR

ROUTINE EnableInFalse   (* ladder *)
// Out of Service is asserted; Outputs OFF; Run Status shown but Alarms inhibited
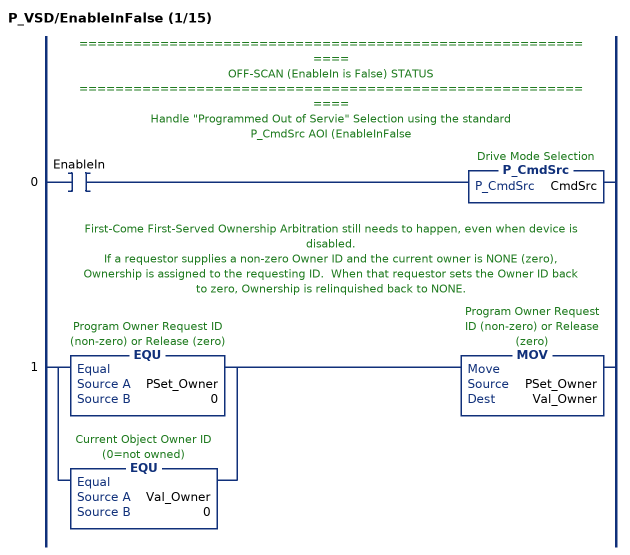
   // ============================================================
   // OFF-SCAN (EnableIn is False) STATUS
   // ============================================================
   // Handle "Programmed Out of Servie" Selection using the standard
   // P_CmdSrc AOI (EnableInFalse
   0: XIC(EnableIn)P_CmdSrc(CmdSrc);
   // First-Come First-Served Ownership Arbitration still needs to happen, even when device is disabled.
   // If a requestor supplies a non-zero Owner ID and the current owner is NONE (zero),
   // Ownership is assigned to the requesting ID.  When that requestor sets the Owner ID back
   // to zero, Ownership is relinquished back to NONE.
   1: [EQU(PSet_Owner,0) ,EQU(Val_Owner,0) ]MOV(PSet_Owner,Val_Owner);
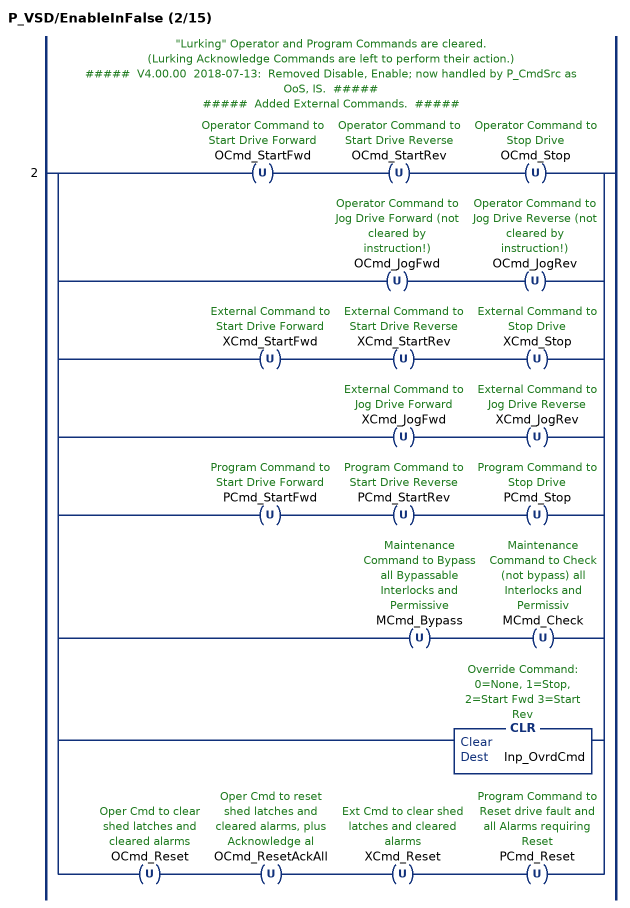
   // "Lurking" Operator and Program Commands are cleared.
   // (Lurking Acknowledge Commands are left to perform their action.)
   // #####  V4.00.00  2018-07-13:  Removed Disable, Enable; now handled by P_CmdSrc as OoS, IS.  #####
   // #####  Added External Commands.  #####
   2: [OTU(OCmd_StartFwd) OTU(OCmd_StartRev) OTU(OCmd_Stop) ,OTU(OCmd_JogFwd) OTU(OCmd_JogRev) ,OTU(XCmd_StartFwd) OTU(XCmd_StartRev) OTU(XCmd_Stop) ,OTU(XCmd_JogFwd) OTU(XCmd_JogRev) ,OTU(PCmd_StartFwd) OTU(PCmd_StartRev) OTU(PCmd_Stop) ,OTU(MCmd_Bypass) OTU(MCmd_Check) ,CLR(Inp_OvrdCmd) ,OTU(OCmd_Reset) OTU(OCmd_ResetAckAll) OTU(XCmd_Reset) OTU(PCmd_Reset) ];
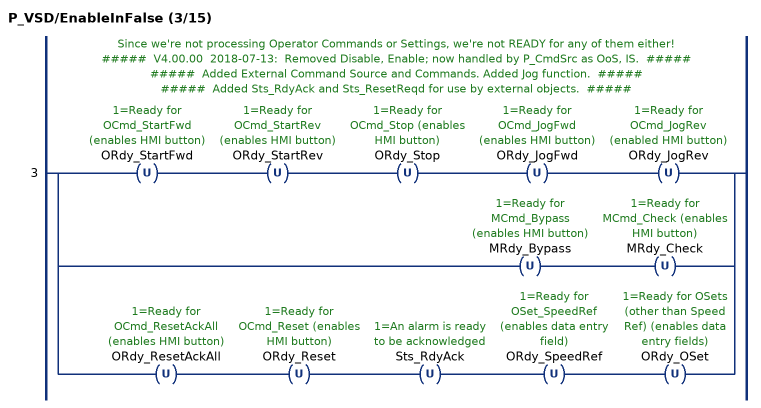
   // Since we're not processing Operator Commands or Settings, we're not READY for any of them either!
   // #####  V4.00.00  2018-07-13:  Removed Disable, Enable; now handled by P_CmdSrc as OoS, IS.  #####
   // #####  Added External Command Source and Commands. Added Jog function.  #####
   // #####  Added Sts_RdyAck and Sts_ResetReqd for use by external objects.  #####
   3: [OTU(ORdy_StartFwd) OTU(ORdy_StartRev) OTU(ORdy_Stop) OTU(ORdy_JogFwd) OTU(ORdy_JogRev) ,OTU(MRdy_Bypass) OTU(MRdy_Check) ,OTU(ORdy_ResetAckAll) OTU(ORdy_Reset) OTU(Sts_RdyAck) OTU(ORdy_SpeedRef) OTU(ORdy_OSet) ];
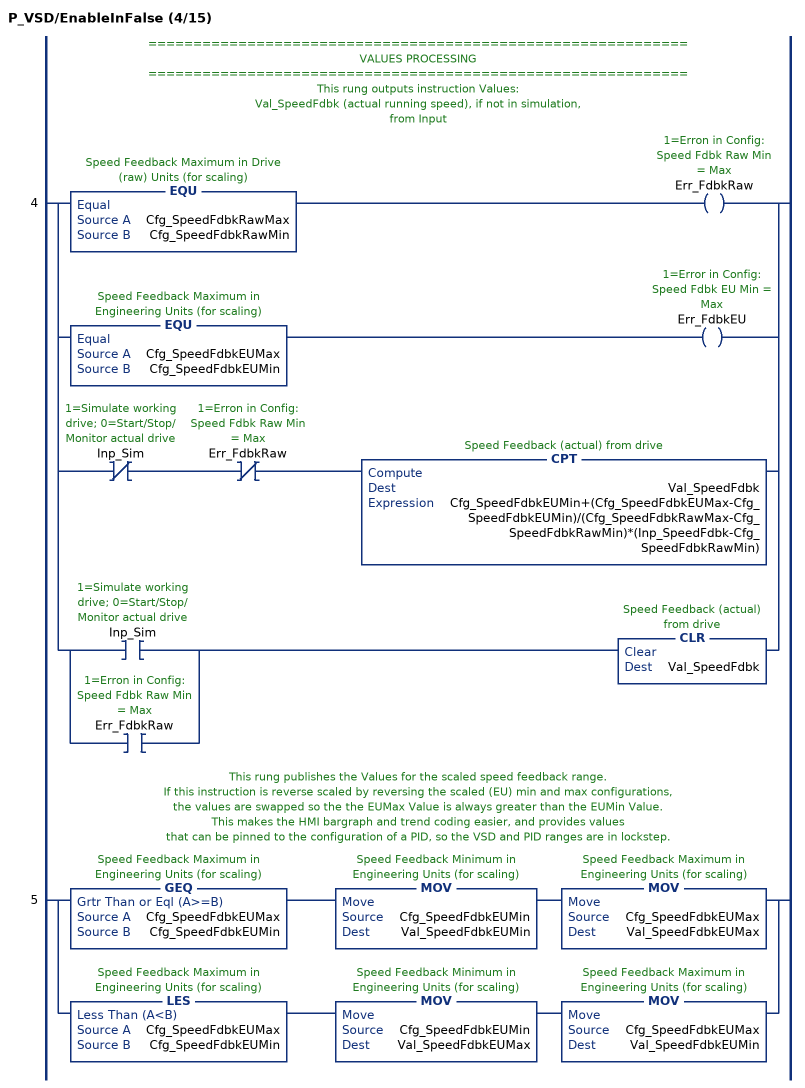
   // ============================================================
   // VALUES PROCESSING
   // ============================================================
   // This rung outputs instruction Values:
   // Val_SpeedFdbk (actual running speed), if not in simulation,
   // from Input
   4: [[EQU(Cfg_SpeedFdbkRawMax,Cfg_SpeedFdbkRawMin) OTE(Err_FdbkRaw) ,EQU(Cfg_SpeedFdbkEUMax,Cfg_SpeedFdbkEUMin) OTE(Err_FdbkEU) ] ,XIO(Inp_Sim) XIO(Err_FdbkRaw) CPT(Val_SpeedFdbk,Cfg_SpeedFdbkEUMin+(Cfg_SpeedFdbkEUMax-Cfg_SpeedFdbkEUMin)/(Cfg_SpeedFdbkRawMax-Cfg_SpeedFdbkRawMin)*(Inp_SpeedFdbk-Cfg_SpeedFdbkRawMin)) ,[XIC(Inp_Sim) ,XIC(Err_FdbkRaw) ] CLR(Val_SpeedFdbk) ];
   // This rung publishes the Values for the scaled speed feedback range.
   // If this instruction is reverse scaled by reversing the scaled (EU) min and max configurations,
   // the values are swapped so the the EUMax Value is always greater than the EUMin Value.
   // This makes the HMI bargraph and trend coding easier, and provides values
   // that can be pinned to the configuration of a PID, so the VSD and PID ranges are in lockstep.
   5: [GEQ(Cfg_SpeedFdbkEUMax,Cfg_SpeedFdbkEUMin) MOV(Cfg_SpeedFdbkEUMin,Val_SpeedFdbkEUMin) MOV(Cfg_SpeedFdbkEUMax,Val_SpeedFdbkEUMax) ,LES(Cfg_SpeedFdbkEUMax,Cfg_SpeedFdbkEUMin) MOV(Cfg_SpeedFdbkEUMin,Val_SpeedFdbkEUMax) MOV(Cfg_SpeedFdbkEUMax,Val_SpeedFdbkEUMin) ];
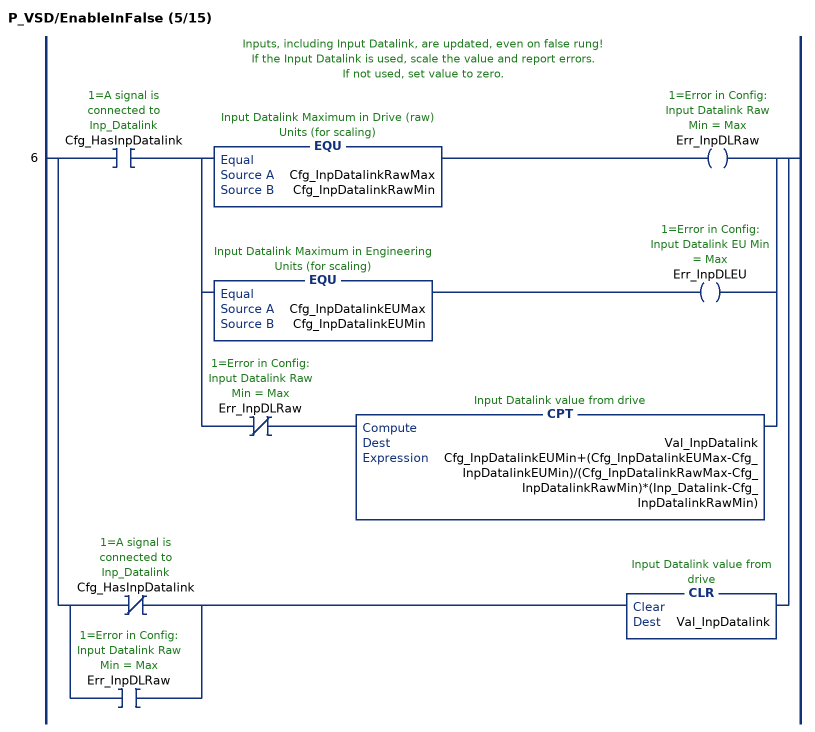
   // Inputs, including Input Datalink, are updated, even on false rung!
   // If the Input Datalink is used, scale the value and report errors.
   // If not used, set value to zero.
   6: [XIC(Cfg_HasInpDatalink) [[EQU(Cfg_InpDatalinkRawMax,Cfg_InpDatalinkRawMin) OTE(Err_InpDLRaw) ,EQU(Cfg_InpDatalinkEUMax,Cfg_InpDatalinkEUMin) OTE(Err_InpDLEU) ] ,XIO(Err_InpDLRaw) CPT(Val_InpDatalink,Cfg_InpDatalinkEUMin+(Cfg_InpDatalinkEUMax-Cfg_InpDatalinkEUMin)/(Cfg_InpDatalinkRawMax-Cfg_InpDatalinkRawMin)*(Inp_Datalink-Cfg_InpDatalinkRawMin)) ] ,[XIO(Cfg_HasInpDatalink) ,XIC(Err_InpDLRaw) ] CLR(Val_InpDatalink) ];
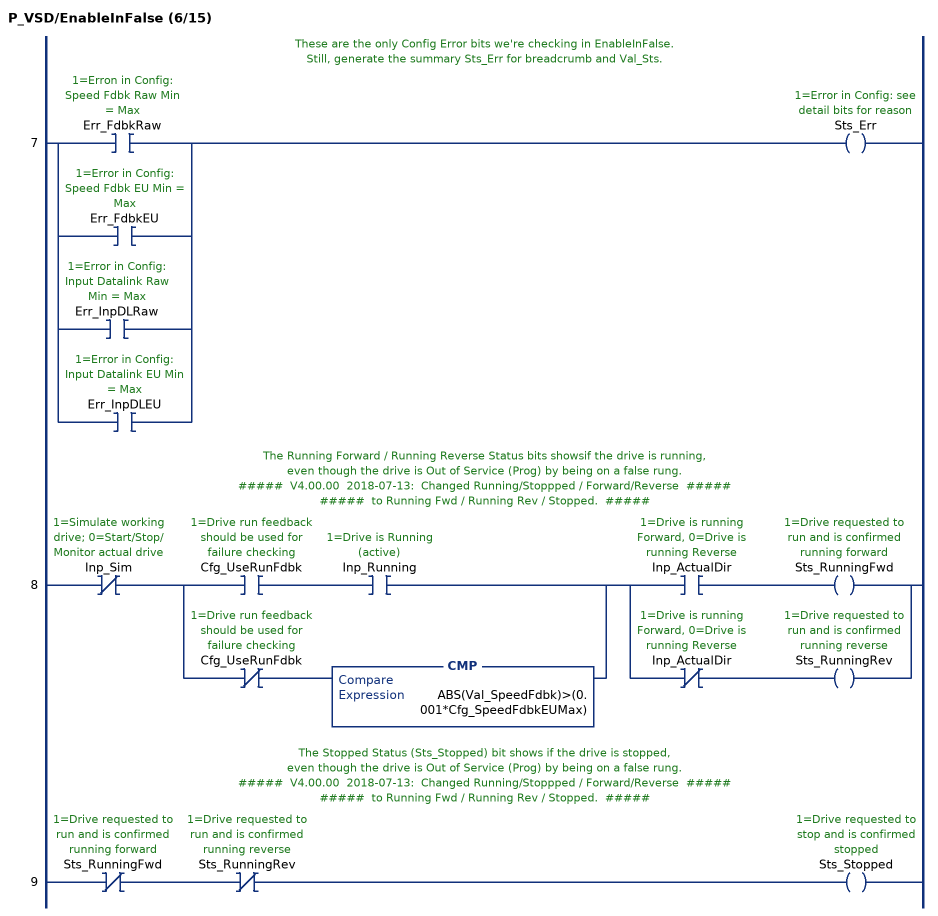
   // These are the only Config Error bits we're checking in EnableInFalse.
   // Still, generate the summary Sts_Err for breadcrumb and Val_Sts.
   7: [XIC(Err_FdbkRaw) ,XIC(Err_FdbkEU) ,XIC(Err_InpDLRaw) ,XIC(Err_InpDLEU) ]OTE(Sts_Err);
   // The Running Forward / Running Reverse Status bits showsif the drive is running,
   // even though the drive is Out of Service (Prog) by being on a false rung.
   // #####  V4.00.00  2018-07-13:  Changed Running/Stoppped / Forward/Reverse  #####
   // #####  to Running Fwd / Running Rev / Stopped.  #####
   8: XIO(Inp_Sim)[XIC(Cfg_UseRunFdbk) XIC(Inp_Running) ,XIO(Cfg_UseRunFdbk) CMP(ABS(Val_SpeedFdbk)>(0.001*Cfg_SpeedFdbkEUMax)) ][XIC(Inp_ActualDir) OTE(Sts_RunningFwd) ,XIO(Inp_ActualDir) OTE(Sts_RunningRev) ];
   // The Stopped Status (Sts_Stopped) bit shows if the drive is stopped,
   // even though the drive is Out of Service (Prog) by being on a false rung.
   // #####  V4.00.00  2018-07-13:  Changed Running/Stoppped / Forward/Reverse  #####
   // #####  to Running Fwd / Running Rev / Stopped.  #####
   9: XIO(Sts_RunningFwd)XIO(Sts_RunningRev)OTE(Sts_Stopped);
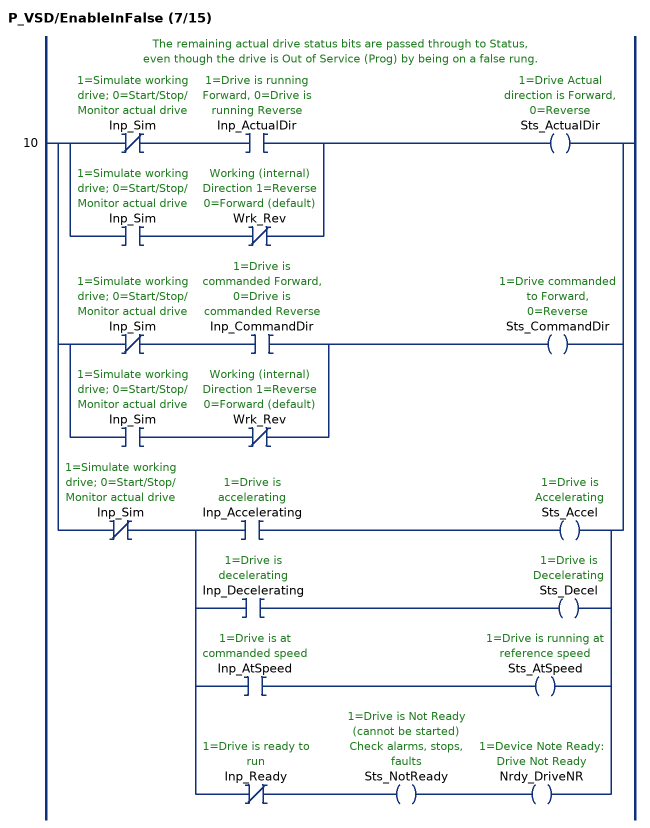
   // The remaining actual drive status bits are passed through to Status,
   // even though the drive is Out of Service (Prog) by being on a false rung.
   10: [[XIO(Inp_Sim) XIC(Inp_ActualDir) ,XIC(Inp_Sim) XIO(Wrk_Rev) ] OTE(Sts_ActualDir) ,[XIO(Inp_Sim) XIC(Inp_CommandDir) ,XIC(Inp_Sim) XIO(Wrk_Rev) ] OTE(Sts_CommandDir) ,XIO(Inp_Sim) [XIC(Inp_Accelerating) OTE(Sts_Accel) ,XIC(Inp_Decelerating) OTE(Sts_Decel) ,XIC(Inp_AtSpeed) OTE(Sts_AtSpeed) ,XIO(Inp_Ready) OTE(Sts_NotReady) OTE(Nrdy_DriveNR) ] ];
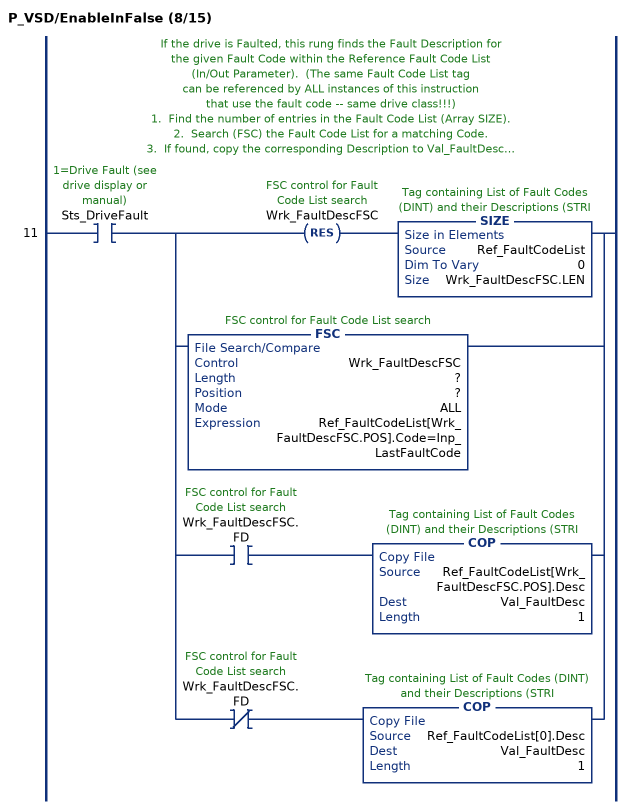
   // If the drive is Faulted, this rung finds the Fault Description for
   // the given Fault Code within the Reference Fault Code List
   // (In/Out Parameter).  (The same Fault Code List tag
   // can be referenced by ALL instances of this instruction
   // that use the fault code -- same drive class!!!)
   // 1.  Find the number of entries in the Fault Code List (Array SIZE).
   // 2.  Search (FSC) the Fault Code List for a matching Code.
   // 3.  If found, copy the corresponding Description to Val_FaultDesc.
   // 4.  If NOT found, copy list entry zero ("No Help Available for this code").
   11: XIC(Sts_DriveFault)[RES(Wrk_FaultDescFSC) SIZE(Ref_FaultCodeList,0,Wrk_FaultDescFSC.LEN) ,FSC(Wrk_FaultDescFSC,?,?,ALL,Ref_FaultCodeList[Wrk_FaultDescFSC.POS].Code=Inp_LastFaultCode) ,XIC(Wrk_FaultDescFSC.FD) COP(Ref_FaultCodeList[Wrk_FaultDescFSC.POS].Desc,Val_FaultDesc,1) ,XIO(Wrk_FaultDescFSC.FD) COP(Ref_FaultCodeList[0].Desc,Val_FaultDesc,1) ];
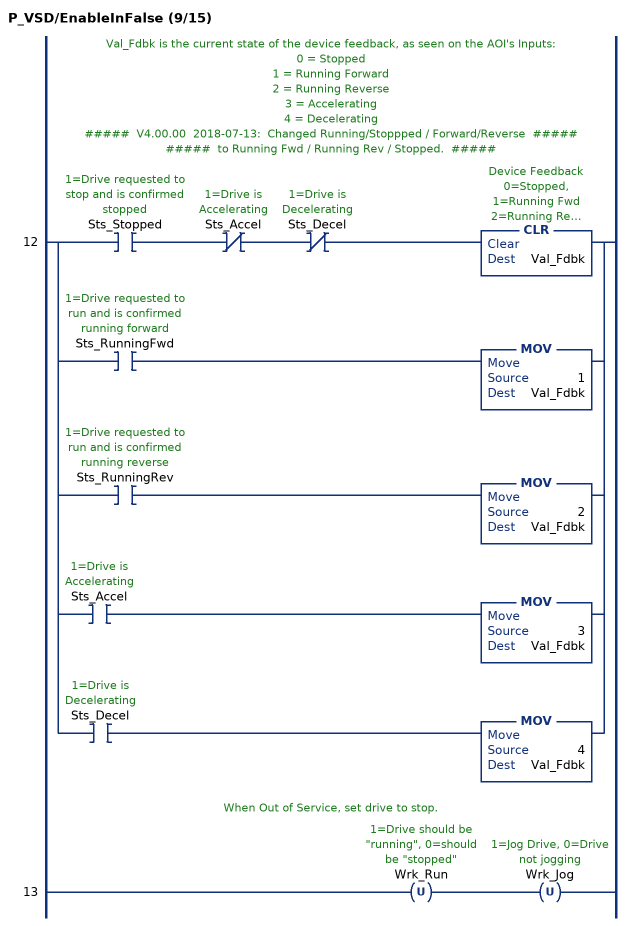
   // Val_Fdbk is the current state of the device feedback, as seen on the AOI's Inputs:
   // 0 = Stopped
   // 1 = Running Forward
   // 2 = Running Reverse
   // 3 = Accelerating
   // 4 = Decelerating
   // #####  V4.00.00  2018-07-13:  Changed Running/Stoppped / Forward/Reverse  #####
   // #####  to Running Fwd / Running Rev / Stopped.  #####
   12: [XIC(Sts_Stopped) XIO(Sts_Accel) XIO(Sts_Decel) CLR(Val_Fdbk) ,XIC(Sts_RunningFwd) MOV(1,Val_Fdbk) ,XIC(Sts_RunningRev) MOV(2,Val_Fdbk) ,XIC(Sts_Accel) MOV(3,Val_Fdbk) ,XIC(Sts_Decel) MOV(4,Val_Fdbk) ];
   // When Out of Service, set drive to stop.
   13: OTU(Wrk_Run)OTU(Wrk_Jog);
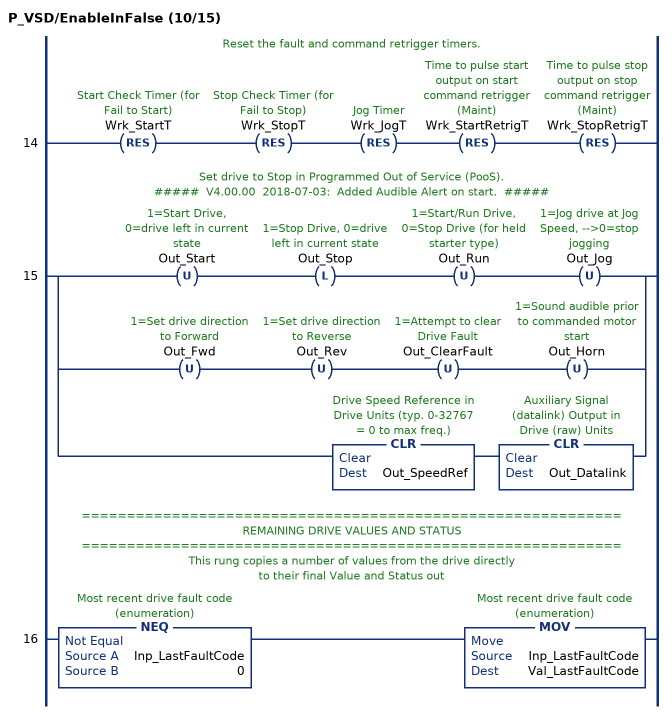
   // Reset the fault and command retrigger timers.
   14: RES(Wrk_StartT)RES(Wrk_StopT)RES(Wrk_JogT)RES(Wrk_StartRetrigT)RES(Wrk_StopRetrigT);
   // Set drive to Stop in Programmed Out of Service (PooS).
   // #####  V4.00.00  2018-07-03:  Added Audible Alert on start.  #####
   15: [OTU(Out_Start) OTL(Out_Stop) OTU(Out_Run) OTU(Out_Jog) ,OTU(Out_Fwd) OTU(Out_Rev) OTU(Out_ClearFault) OTU(Out_Horn) ,CLR(Out_SpeedRef) CLR(Out_Datalink) ];
   // ============================================================
   // REMAINING DRIVE VALUES AND STATUS
   // ============================================================
   // This rung copies a number of values from the drive directly
   // to their final Value and Status out
   16: NEQ(Inp_LastFaultCode,0)MOV(Inp_LastFaultCode,Val_LastFaultCode);
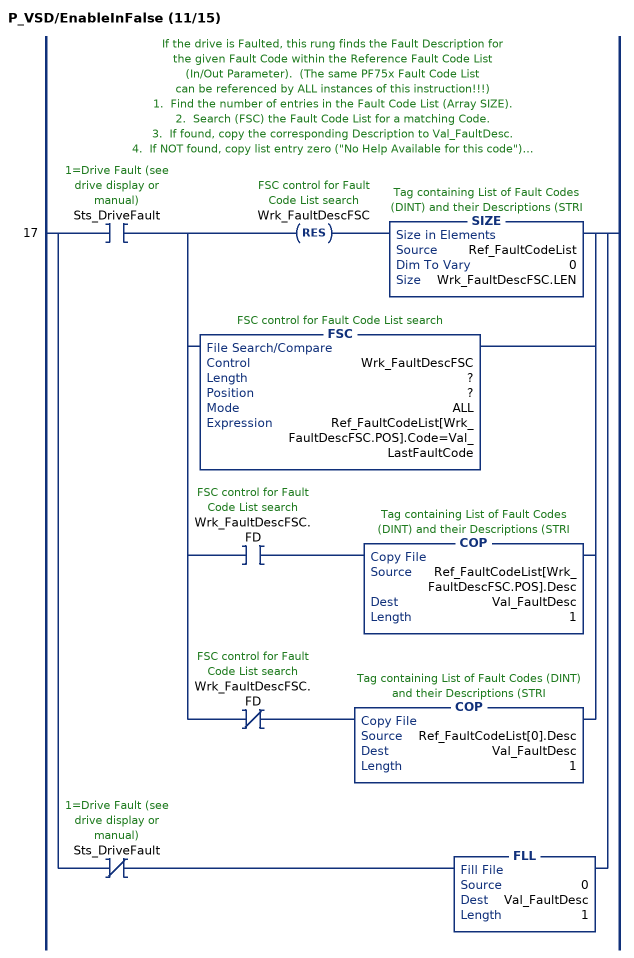
   // If the drive is Faulted, this rung finds the Fault Description for
   // the given Fault Code within the Reference Fault Code List
   // (In/Out Parameter).  (The same PF75x Fault Code List
   // can be referenced by ALL instances of this instruction!!!)
   // 1.  Find the number of entries in the Fault Code List (Array SIZE).
   // 2.  Search (FSC) the Fault Code List for a matching Code.
   // 3.  If found, copy the corresponding Description to Val_FaultDesc.
   // 4.  If NOT found, copy list entry zero ("No Help Available for this code").
   // And if the drive is not faulted, clear the Val_FaultDesc string.
   17: [XIC(Sts_DriveFault) [RES(Wrk_FaultDescFSC) SIZE(Ref_FaultCodeList,0,Wrk_FaultDescFSC.LEN) ,FSC(Wrk_FaultDescFSC,?,?,ALL,Ref_FaultCodeList[Wrk_FaultDescFSC.POS].Code=Val_LastFaultCode) ,XIC(Wrk_FaultDescFSC.FD) COP(Ref_FaultCodeList[Wrk_FaultDescFSC.POS].Desc,Val_FaultDesc,1) ,XIO(Wrk_FaultDescFSC.FD) COP(Ref_FaultCodeList[0].Desc,Val_FaultDesc,1) ] ,XIO(Sts_DriveFault) FLL(0,Val_FaultDesc,1) ];
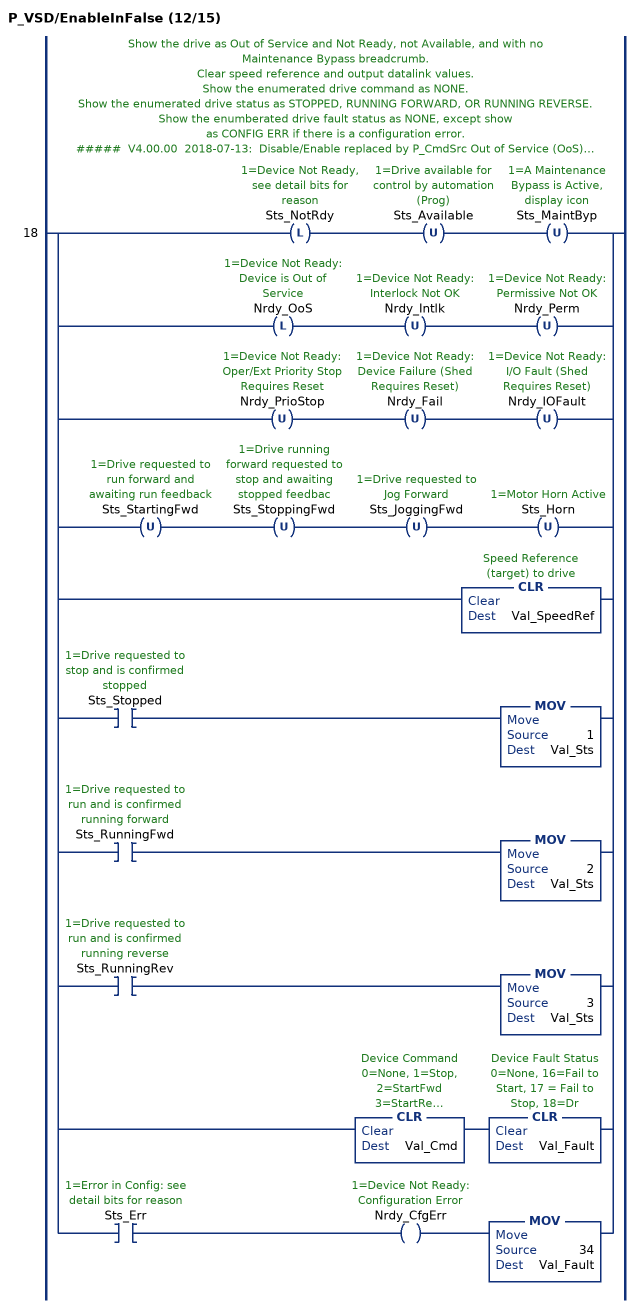
   // Show the drive as Out of Service and Not Ready, not Available, and with no
   // Maintenance Bypass breadcrumb.
   // Clear speed reference and output datalink values.
   // Show the enumerated drive command as NONE.
   // Show the enumerated drive status as STOPPED, RUNNING FORWARD, OR RUNNING REVERSE.
   // Show the enumberated drive fault status as NONE, except show
   // as CONFIG ERR if there is a configuration error.
   // #####  V4.00.00  2018-07-13:  Disable/Enable replaced by P_CmdSrc Out of Service (OoS).  #####
   // #####  Updated Val_Sts to common enumeration across all motors and drives.  #####
   18: [OTL(Sts_NotRdy) OTU(Sts_Available) OTU(Sts_MaintByp) ,OTL(Nrdy_OoS) OTU(Nrdy_Intlk) OTU(Nrdy_Perm) ,OTU(Nrdy_PrioStop) OTU(Nrdy_Fail) OTU(Nrdy_IOFault) ,OTU(Sts_StartingFwd) OTU(Sts_StoppingFwd) OTU(Sts_JoggingFwd) OTU(Sts_Horn) ,CLR(Val_SpeedRef) ,XIC(Sts_Stopped) MOV(1,Val_Sts) ,XIC(Sts_RunningFwd) MOV(2,Val_Sts) ,XIC(Sts_RunningRev) MOV(3,Val_Sts) ,CLR(Val_Cmd) CLR(Val_Fault) ,XIC(Sts_Err) OTE(Nrdy_CfgErr) MOV(34,Val_Fault) ];
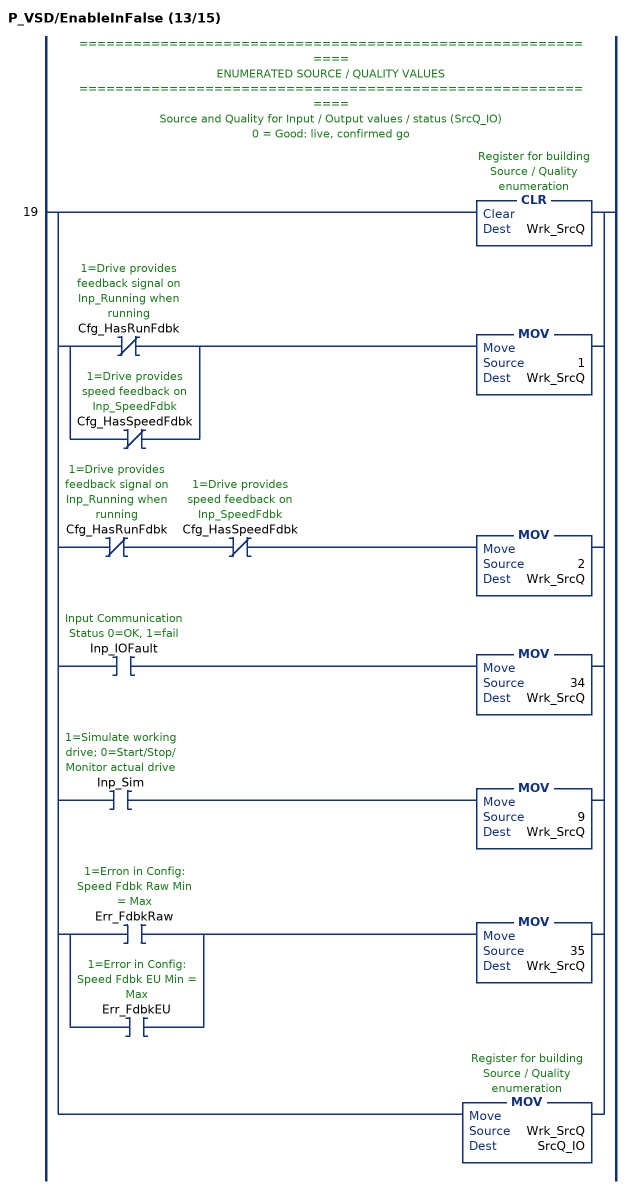
   // ============================================================
   // ENUMERATED SOURCE / QUALITY VALUES
   // ============================================================
   // Source and Quality for Input / Output values / status (SrcQ_IO)
   // 0 = Good: live, confirmed go
   19: [CLR(Wrk_SrcQ) ,[XIO(Cfg_HasRunFdbk) ,XIO(Cfg_HasSpeedFdbk) ] MOV(1,Wrk_SrcQ) ,XIO(Cfg_HasRunFdbk) XIO(Cfg_HasSpeedFdbk) MOV(2,Wrk_SrcQ) ,XIC(Inp_IOFault) MOV(34,Wrk_SrcQ) ,XIC(Inp_Sim) MOV(9,Wrk_SrcQ) ,[XIC(Err_FdbkRaw) ,XIC(Err_FdbkEU) ] MOV(35,Wrk_SrcQ) ,MOV(Wrk_SrcQ,SrcQ_IO) ];
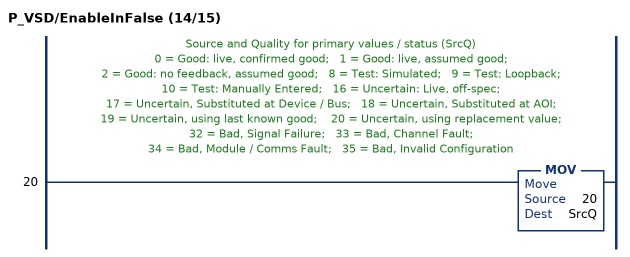
   // Source and Quality for primary values / status (SrcQ)
   // 0 = Good: live, confirmed good;   1 = Good: live, assumed good;
   // 2 = Good: no feedback, assumed good;   8 = Test: Simulated;   9 = Test: Loopback;
   // 10 = Test: Manually Entered;   16 = Uncertain: Live, off-spec;
   // 17 = Uncertain, Substituted at Device / Bus;   18 = Uncertain, Substituted at AOI;
   // 19 = Uncertain, using last known good;    20 = Uncertain, using replacement value;
   // 32 = Bad, Signal Failure;   33 = Bad, Channel Fault;
   // 34 = Bad, Module / Comms Fault;   35 = Bad, Invalid Configuration
   20: MOV(20,SrcQ);
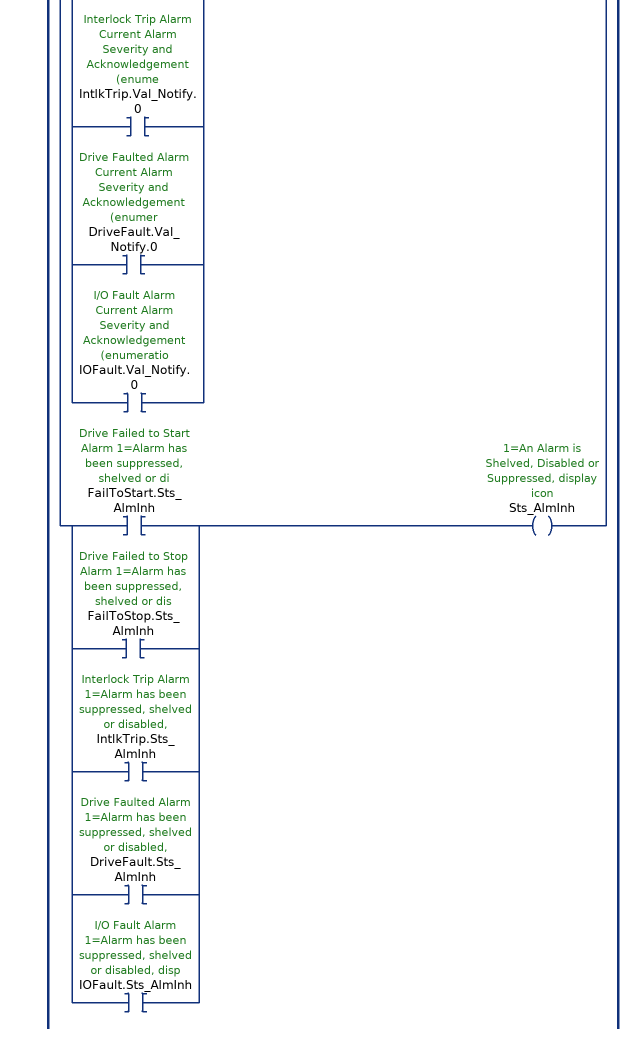
   // If the device is OFF-SCAN (rung is false or EnableIn is false in FBD),
   // then show the alarms as "Parent object out of service".
   // Show the overall acknowledgement status.
   // #####  V4.00.00  2018-07-13:  Changed P_Mode to P_CmdSrc, added Out of Service.  #####
   21: [OTL(FailToStart.Inp_OoS) P_Alarm(FailToStart) ,OTL(FailToStop.Inp_OoS) P_Alarm(FailToStop) ,OTL(IntlkTrip.Inp_OoS) P_Alarm(IntlkTrip) ,OTL(DriveFault.Inp_OoS) P_Alarm(DriveFault) ,OTL(IOFault.Inp_OoS) P_Alarm(IOFault) ,CLR(Val_Notify) CLR(Val_NotifyAll) ,[XIC(FailToStart.Val_Notify.0) ,XIC(FailToStop.Val_Notify.0) ,XIC(IntlkTrip.Val_Notify.0) ,XIC(DriveFault.Val_Notify.0) ,XIC(IOFault.Val_Notify.0) ] OTL(Val_Notify.0) OTL(Val_NotifyAll.0) ,[XIC(FailToStart.Sts_AlmInh) ,XIC(FailToStop.Sts_AlmInh) ,XIC(IntlkTrip.Sts_AlmInh) ,XIC(DriveFault.Sts_AlmInh) ,XIC(IOFault.Sts_AlmInh) ] OTE(Sts_AlmInh) ];
END_ROUTINE

ROUTINE Logic   (* ladder *)
// Normal Scan: control / monitor Variable-Speed Drive
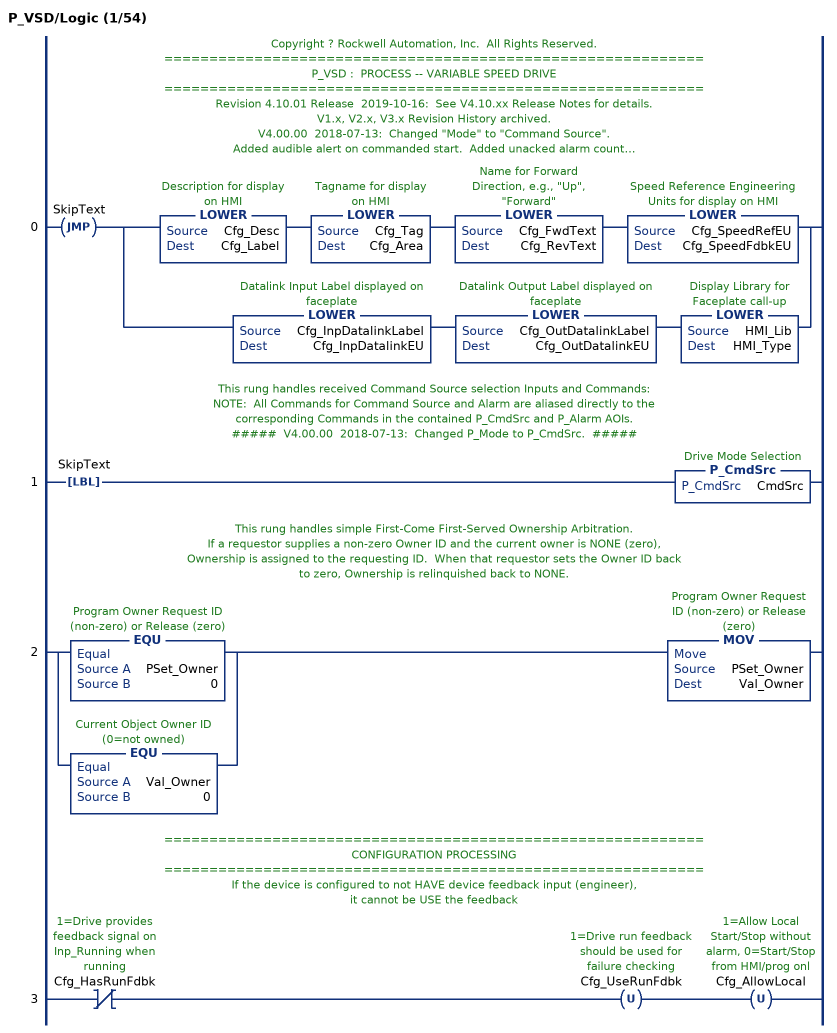
   // Copyright ? Rockwell Automation, Inc.  All Rights Reserved.
   // ============================================================
   // P_VSD :  PROCESS -- VARIABLE SPEED DRIVE
   // ============================================================
   // Revision 4.10.01 Release  2019-10-16:  See V4.10.xx Release Notes for details.
   // V1.x, V2.x, V3.x Revision History archived.
   // V4.00.00  2018-07-13:  Changed "Mode" to "Command Source".
   // Added audible alert on commanded start.  Added unacked alarm count.
   // Changed Inf_ items to HMI_, and added Cfg_Area for security.
   // Changed Start / Stop / Fwd / Rev / Jog to StartFwd / StartRev /Stop / JogFwd / JogRev.
   // Deleted Cfg_PCmdClear; all Program Commands are now self-clearing.
   // All OCmds/MCmds and ORdys/MRdys are now Local Tags.
   // Added Sts_RdyAck and Sts_ResetReqd for use by external objects.
   // Aligned ready bit naming with command bit names.
   // Added configurable decimal places for display on HMI.
   // Modifications to Output Datalink clamp limit restrictions / checking.
   // Changed delay / time configuration items to REAL seconds.
   // Updated Val_Sts to common enumeration across all motors and drives.
   // V4.00.02  2018-10-30:  Corrected handling Allow Local when horn is enabled
   // V4.10.00  2019-03-25:  Changed availability to use input availability from interlocks.
   // Added Horn Status, Horn Inhibit. Updated to P_CmdSrc V4.10.00.
   // Modified simulated run feedback to handle run at zero speed ref.
   // Added Cfg_HasMoreObj.
   // V4.10.01  2019-10-16:  Corrected handling of Start Horn on shed conditions.
   // Modified to lock out jog when jog time expires until jog commands
   // are cleared. Modified to handle overlapping Horn and Jog times.
   // ============================================================
   // This Instruction controls and monitors a Variable-Speed Drive (AC or DC) and provides:
   // *  Starting, stopping, jogging of drive, setting speed reference and direction
   // *  Monitoring of run feedback, display of actual drive status, including accel, decel, direction, speed
   // *  Detection of Failure to Start, Failure to Stop, Drive Fault
   // *  Monitoring of Permissive conditions to allow starting
   // * Monitoring of Interlock conditions to stop / prevent starting
   // * Simulation, providing feedback of a working drive while disabling outputs
   // * Monitoring of I/O communication faults
   // * Alarms for Fail to Start, Fail to Stop, Interlock Trip, Drive Fault, I/O Fault
   // * Option to automatically reset faults and alarms when operator commands
   // motor to start or stop
   // * Supports HMI "breadcrumbs" for Alarm Inhibited, Bad Configuration,
   // Not Ready, Maintenance Bypass Active
   // * "Available" status for use by automation logic to know whether motor
   // can be controlled by other objects.
   // * Horn output for audible alert prior to starting motor.
   // Command Sources are arbitrated by a P_CmdSrc Add-On Instruction instance.
   // Command Sources: Operator, External, Program, External, Override, Maintenance,
   // Out of Service, Hand.  Alarms are provided by P_Alarm Add-On Instruction instances.
   // ============================================================
   // SHOW LOCAL STRINGS
   // ============================================================
   // The STRINGs containing the text associated with each instance of this
   // instruction cannot be Input or Output Parameters, because STRINGs are not
   //  'atomic' types. (Inputs and Outputs must be SINT, INT, DINT, REAL, or BOOL.)
   // In order to make it easier to find and configure these STRINGs, this rung
   // was added.  THE JMP (and the LBL on the following rung)
   // MUST NOT BE REMOVED!!!
   // To view the STRINGs, go to the instruction instance (in LD or FBD), RIGHT-click
   // to bring up the context menu and select "Open Instruction Logic".
   // This rung will appear with the STRING values for the selected instance.
   // You may double-click the STRING values here to modify them as well.
   // #####  V4.00.00  2018-07-13:  Added string for Cfg_Area, renamed Inf_* to HMI_*.  #####
   0: JMP(SkipText)[LOWER(Cfg_Desc,Cfg_Label) LOWER(Cfg_Tag,Cfg_Area) LOWER(Cfg_FwdText,Cfg_RevText) LOWER(Cfg_SpeedRefEU,Cfg_SpeedFdbkEU) ,LOWER(Cfg_InpDatalinkLabel,Cfg_InpDatalinkEU) LOWER(Cfg_OutDatalinkLabel,Cfg_OutDatalinkEU) LOWER(HMI_Lib,HMI_Type) ];
   // This rung handles received Command Source selection Inputs and Commands:
   // NOTE:  All Commands for Command Source and Alarm are aliased directly to the
   // corresponding Commands in the contained P_CmdSrc and P_Alarm AOIs.
   // #####  V4.00.00  2018-07-13:  Changed P_Mode to P_CmdSrc.  #####
   1: LBL(SkipText)P_CmdSrc(CmdSrc);
   // This rung handles simple First-Come First-Served Ownership Arbitration.
   // If a requestor supplies a non-zero Owner ID and the current owner is NONE (zero),
   // Ownership is assigned to the requesting ID.  When that requestor sets the Owner ID back
   // to zero, Ownership is relinquished back to NONE.
   2: [EQU(PSet_Owner,0) ,EQU(Val_Owner,0) ]MOV(PSet_Owner,Val_Owner);
   // ============================================================
   // CONFIGURATION PROCESSING
   // ============================================================
   // If the device is configured to not HAVE device feedback input (engineer),
   // it cannot be USE the feedback
   3: XIO(Cfg_HasRunFdbk)OTU(Cfg_UseRunFdbk)OTU(Cfg_AllowLocal);
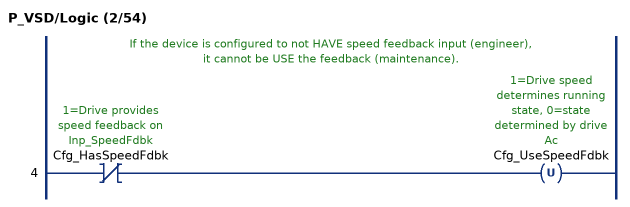
   // If the device is configured to not HAVE speed feedback input (engineer),
   // it cannot be USE the feedback (maintenance).
   4: XIO(Cfg_HasSpeedFdbk)OTU(Cfg_UseSpeedFdbk);
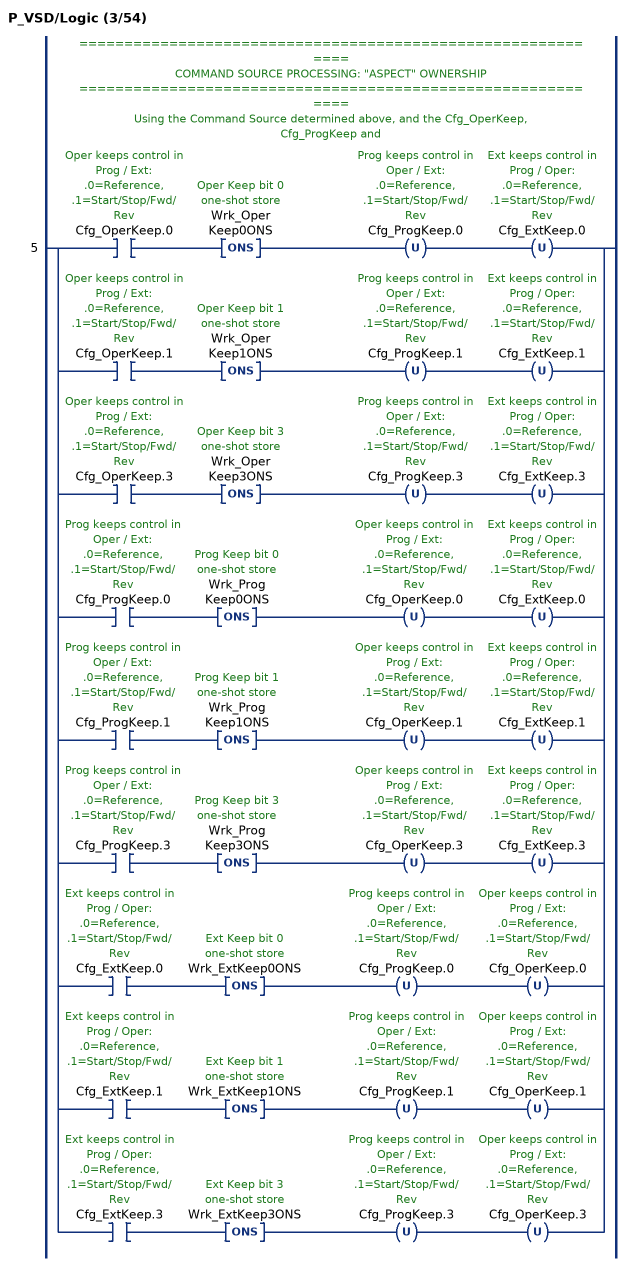
   // ============================================================
   // COMMAND SOURCE PROCESSING: "ASPECT" OWNERSHIP
   // ============================================================
   // Using the Command Source determined above, and the Cfg_OperKeep,
   // Cfg_ProgKeep and
   5: [XIC(Cfg_OperKeep.0) ONS(Wrk_OperKeep0ONS) OTU(Cfg_ProgKeep.0) OTU(Cfg_ExtKeep.0) ,XIC(Cfg_OperKeep.1) ONS(Wrk_OperKeep1ONS) OTU(Cfg_ProgKeep.1) OTU(Cfg_ExtKeep.1) ,XIC(Cfg_OperKeep.3) ONS(Wrk_OperKeep3ONS) OTU(Cfg_ProgKeep.3) OTU(Cfg_ExtKeep.3) ,XIC(Cfg_ProgKeep.0) ONS(Wrk_ProgKeep0ONS) OTU(Cfg_OperKeep.0) OTU(Cfg_ExtKeep.0) ,XIC(Cfg_ProgKeep.1) ONS(Wrk_ProgKeep1ONS) OTU(Cfg_OperKeep.1) OTU(Cfg_ExtKeep.1) ,XIC(Cfg_ProgKeep.3) ONS(Wrk_ProgKeep3ONS) OTU(Cfg_OperKeep.3) OTU(Cfg_ExtKeep.3) ,XIC(Cfg_ExtKeep.0) ONS(Wrk_ExtKeep0ONS) OTU(Cfg_ProgKeep.0) OTU(Cfg_OperKeep.0) ,XIC(Cfg_ExtKeep.1) ONS(Wrk_ExtKeep1ONS) OTU(Cfg_ProgKeep.1) OTU(Cfg_OperKeep.1) ,XIC(Cfg_ExtKeep.3) ONS(Wrk_ExtKeep3ONS) OTU(Cfg_ProgKeep.3) OTU(Cfg_OperKeep.3) ];
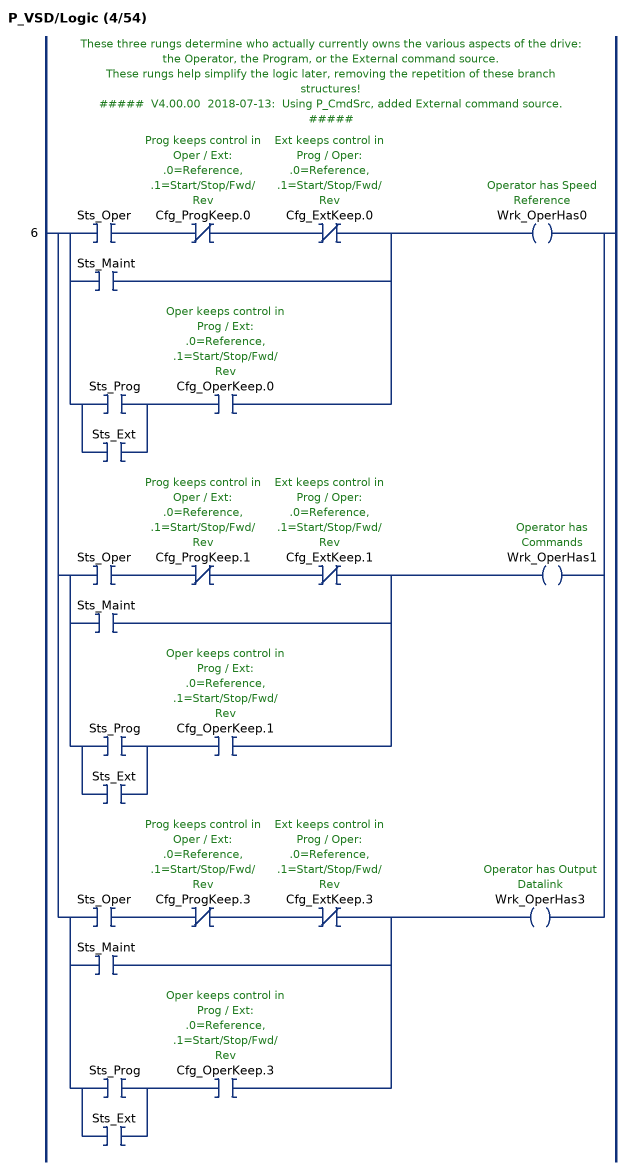
   // These three rungs determine who actually currently owns the various aspects of the drive:
   // the Operator, the Program, or the External command source.
   // These rungs help simplify the logic later, removing the repetition of these branch structures!
   // #####  V4.00.00  2018-07-13:  Using P_CmdSrc, added External command source.  #####
   6: [[XIC(Sts_Oper) XIO(Cfg_ProgKeep.0) XIO(Cfg_ExtKeep.0) ,XIC(Sts_Maint) ,[XIC(Sts_Prog) ,XIC(Sts_Ext) ] XIC(Cfg_OperKeep.0) ] OTE(Wrk_OperHas0) ,[XIC(Sts_Oper) XIO(Cfg_ProgKeep.1) XIO(Cfg_ExtKeep.1) ,XIC(Sts_Maint) ,[XIC(Sts_Prog) ,XIC(Sts_Ext) ] XIC(Cfg_OperKeep.1) ] OTE(Wrk_OperHas1) ,[XIC(Sts_Oper) XIO(Cfg_ProgKeep.3) XIO(Cfg_ExtKeep.3) ,XIC(Sts_Maint) ,[XIC(Sts_Prog) ,XIC(Sts_Ext) ] XIC(Cfg_OperKeep.3) ] OTE(Wrk_OperHas3) ];
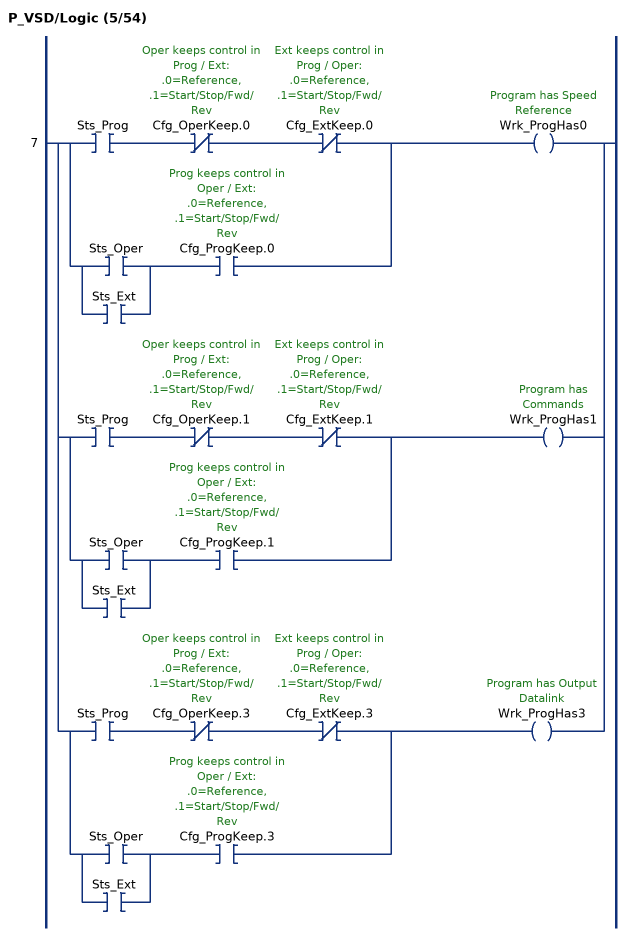
   7: [[XIC(Sts_Prog) XIO(Cfg_OperKeep.0) XIO(Cfg_ExtKeep.0) ,[XIC(Sts_Oper) ,XIC(Sts_Ext) ] XIC(Cfg_ProgKeep.0) ] OTE(Wrk_ProgHas0) ,[XIC(Sts_Prog) XIO(Cfg_OperKeep.1) XIO(Cfg_ExtKeep.1) ,[XIC(Sts_Oper) ,XIC(Sts_Ext) ] XIC(Cfg_ProgKeep.1) ] OTE(Wrk_ProgHas1) ,[XIC(Sts_Prog) XIO(Cfg_OperKeep.3) XIO(Cfg_ExtKeep.3) ,[XIC(Sts_Oper) ,XIC(Sts_Ext) ] XIC(Cfg_ProgKeep.3) ] OTE(Wrk_ProgHas3) ];
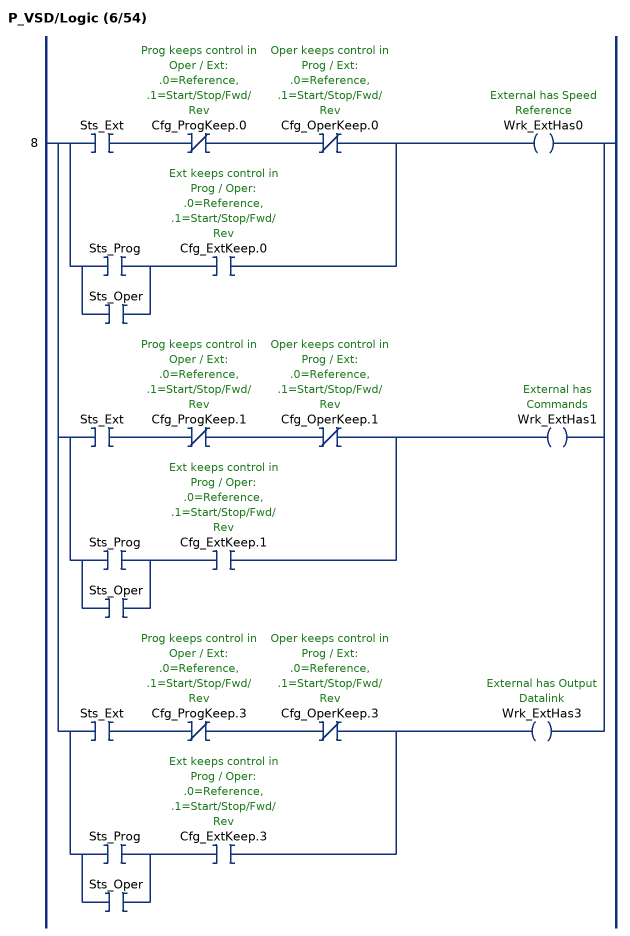
   8: [[XIC(Sts_Ext) XIO(Cfg_ProgKeep.0) XIO(Cfg_OperKeep.0) ,[XIC(Sts_Prog) ,XIC(Sts_Oper) ] XIC(Cfg_ExtKeep.0) ] OTE(Wrk_ExtHas0) ,[XIC(Sts_Ext) XIO(Cfg_ProgKeep.1) XIO(Cfg_OperKeep.1) ,[XIC(Sts_Prog) ,XIC(Sts_Oper) ] XIC(Cfg_ExtKeep.1) ] OTE(Wrk_ExtHas1) ,[XIC(Sts_Ext) XIO(Cfg_ProgKeep.3) XIO(Cfg_OperKeep.3) ,[XIC(Sts_Prog) ,XIC(Sts_Oper) ] XIC(Cfg_ExtKeep.3) ] OTE(Wrk_ExtHas3) ];
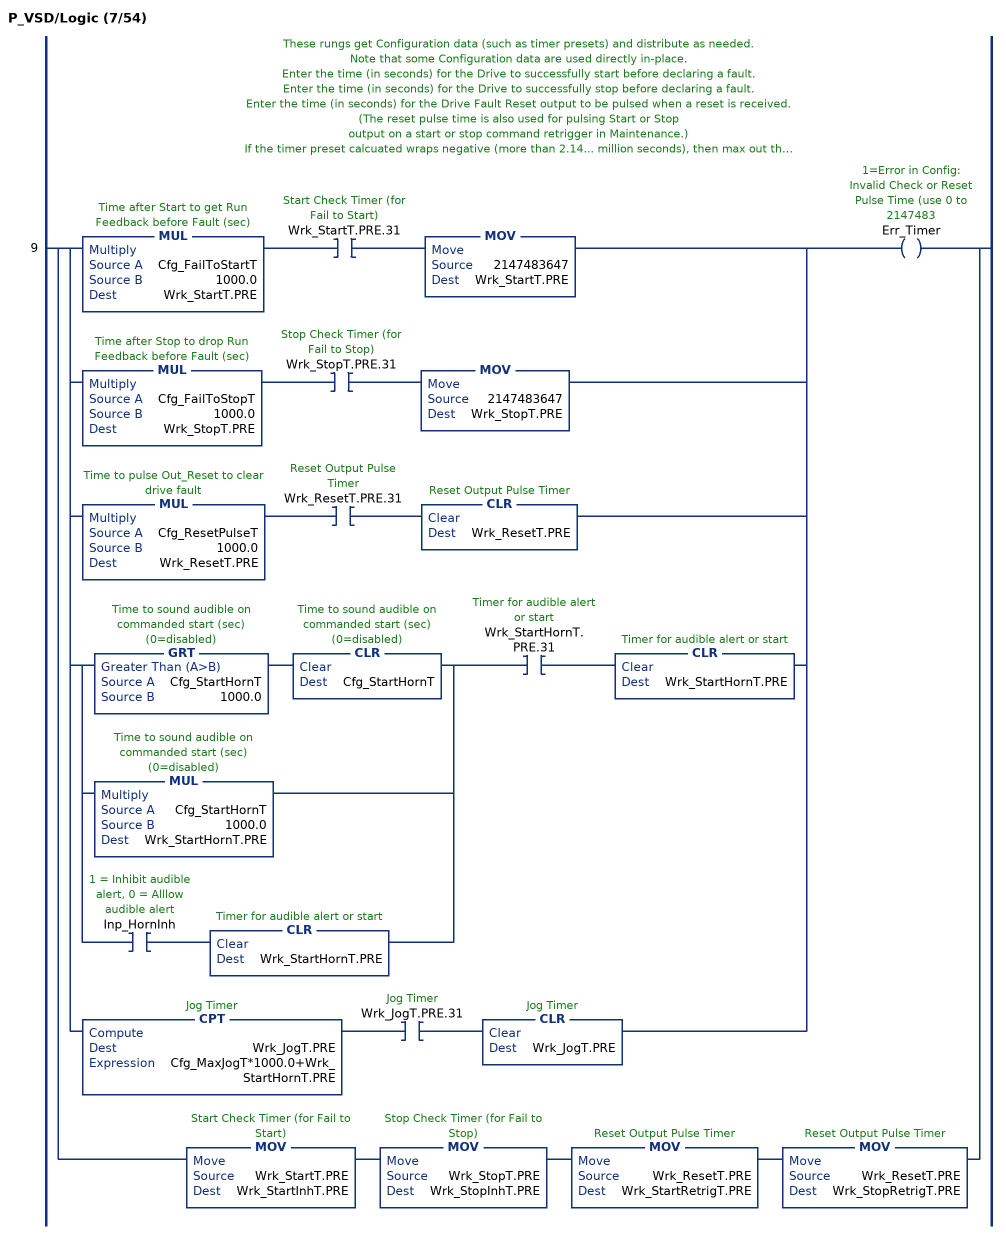
   // These rungs get Configuration data (such as timer presets) and distribute as needed.
   // Note that some Configuration data are used directly in-place.
   // Enter the time (in seconds) for the Drive to successfully start before declaring a fault.
   // Enter the time (in seconds) for the Drive to successfully stop before declaring a fault.
   // Enter the time (in seconds) for the Drive Fault Reset output to be pulsed when a reset is received.
   // (The reset pulse time is also used for pulsing Start or Stop
   // output on a start or stop command retrigger in Maintenance.)
   // If the timer preset calcuated wraps negative (more than 2.14... million seconds), then max out the
   // or clear the Timer Preset (as appropriate) and flag it.  Note that a negative timer preset will fault the controller!!!
   // #####  V4.00.00  2018-07-13:  Added audible alert prior to commanded start.  #####
   // #####  Changed delay / time configuration items to REAL seconds.  #####
   // #####  V4.10.00  2019-03-25:  Added Inp_HornInh to disable Horn operation.  #####
   // #####  V4.10.01  2019-10-16:  Modified to handle overlapping Horn and Jog times.  #####
   9: [[MUL(Cfg_FailToStartT,1000.0,Wrk_StartT.PRE) XIC(Wrk_StartT.PRE.31) MOV(2147483647,Wrk_StartT.PRE) ,MUL(Cfg_FailToStopT,1000.0,Wrk_StopT.PRE) XIC(Wrk_StopT.PRE.31) MOV(2147483647,Wrk_StopT.PRE) ,MUL(Cfg_ResetPulseT,1000.0,Wrk_ResetT.PRE) XIC(Wrk_ResetT.PRE.31) CLR(Wrk_ResetT.PRE) ,[GRT(Cfg_StartHornT,1000.0) CLR(Cfg_StartHornT) ,MUL(Cfg_StartHornT,1000.0,Wrk_StartHornT.PRE) ,XIC(Inp_HornInh) CLR(Wrk_StartHornT.PRE) ] XIC(Wrk_StartHornT.PRE.31) CLR(Wrk_StartHornT.PRE) ,CPT(Wrk_JogT.PRE,Cfg_MaxJogT*1000.0+Wrk_StartHornT.PRE) XIC(Wrk_JogT.PRE.31) CLR(Wrk_JogT.PRE) ] OTE(Err_Timer) ,MOV(Wrk_StartT.PRE,Wrk_StartInhT.PRE) MOV(Wrk_StopT.PRE,Wrk_StopInhT.PRE) MOV(Wrk_ResetT.PRE,Wrk_StartRetrigT.PRE) MOV(Wrk_ResetT.PRE,Wrk_StopRetrigT.PRE) ];
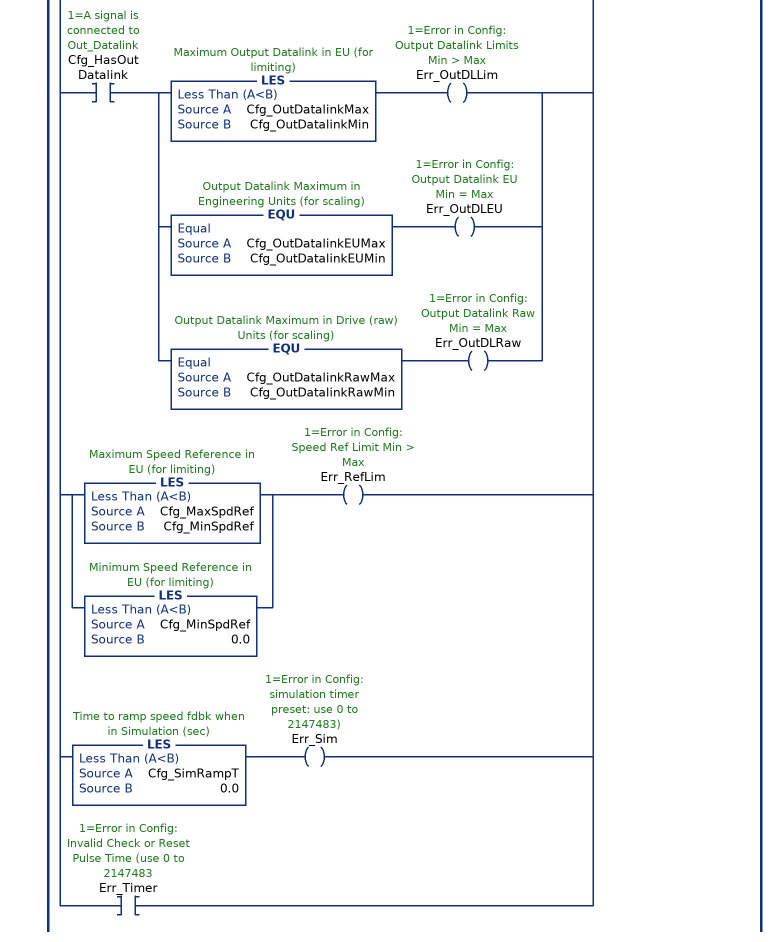
   // This rung handles the reports of all Bad Configuration Status.
   // Individual bits are provided for various status:
   // Bad Raw Scaling configs
   // Bad Engineering Units Scaling configs
   // Bad Min or Max Speed Reference clamp limit
   // Bad simulation speed ramp time
   // Bad timer config from (rung above)
   // Bad Alarm config (from P_Alarm)
   // Bad Cfg_OperKeep / Cfg_ProgKeep config
   // Then a summary Bad Config status is provided, simply an OR of the individual bits.
   // #####  V4.00.00  2018-07-13:  Modified to allow the special case where min and max clamping  #####
   // #####  limits (speed or output datalink) can be EQUAL (clamp at a specific value).  #####
   // #####  Changed delay / time configuration items to REAL seconds.  #####
   10: [XIC(Cfg_HasSpeedFdbk) [EQU(Cfg_SpeedFdbkRawMax,Cfg_SpeedFdbkRawMin) OTE(Err_FdbkRaw) ,EQU(Cfg_SpeedFdbkEUMax,Cfg_SpeedFdbkEUMin) OTE(Err_FdbkEU) ] ,EQU(Cfg_SpeedRefEUMax,Cfg_SpeedRefEUMin) OTE(Err_RefEU) ,EQU(Cfg_SpeedRefRawMax,Cfg_SpeedRefRawMin) OTE(Err_RefRaw) ,XIC(Cfg_HasInpDatalink) [EQU(Cfg_InpDatalinkRawMax,Cfg_InpDatalinkRawMin) OTE(Err_InpDLRaw) ,EQU(Cfg_InpDatalinkEUMax,Cfg_InpDatalinkEUMin) OTE(Err_InpDLEU) ] ,XIC(Cfg_HasOutDatalink) [LES(Cfg_OutDatalinkMax,Cfg_OutDatalinkMin) OTE(Err_OutDLLim) ,EQU(Cfg_OutDatalinkEUMax,Cfg_OutDatalinkEUMin) OTE(Err_OutDLEU) ,EQU(Cfg_OutDatalinkRawMax,Cfg_OutDatalinkRawMin) OTE(Err_OutDLRaw) ] ,[LES(Cfg_MaxSpdRef,Cfg_MinSpdRef) ,LES(Cfg_MinSpdRef,0.0) ] OTE(Err_RefLim) ,LES(Cfg_SimRampT,0.0) OTE(Err_Sim) ,XIC(Err_Timer) ]OTE(Nrdy_CfgErr);
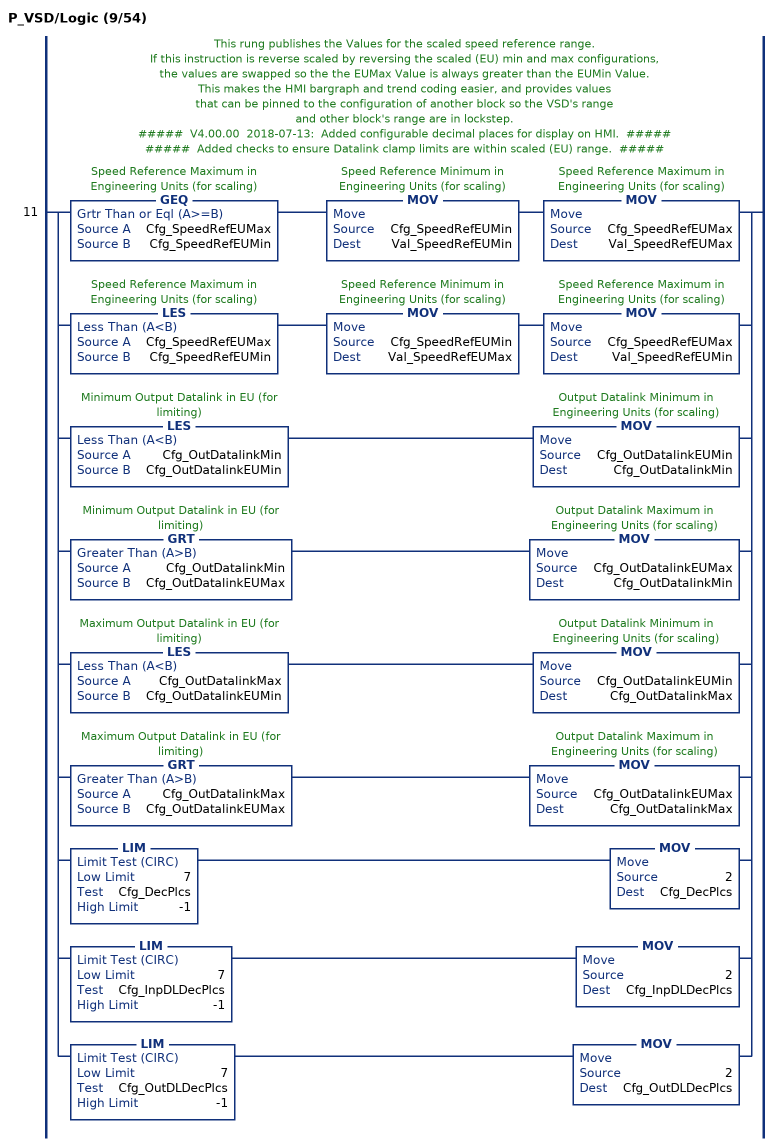
   // This rung publishes the Values for the scaled speed reference range.
   // If this instruction is reverse scaled by reversing the scaled (EU) min and max configurations,
   // the values are swapped so the the EUMax Value is always greater than the EUMin Value.
   // This makes the HMI bargraph and trend coding easier, and provides values
   // that can be pinned to the configuration of another block so the VSD's range
   //  and other block's range are in lockstep.
   // #####  V4.00.00  2018-07-13:  Added configurable decimal places for display on HMI.  #####
   // #####  Added checks to ensure Datalink clamp limits are within scaled (EU) range.  #####
   11: [GEQ(Cfg_SpeedRefEUMax,Cfg_SpeedRefEUMin) MOV(Cfg_SpeedRefEUMin,Val_SpeedRefEUMin) MOV(Cfg_SpeedRefEUMax,Val_SpeedRefEUMax) ,LES(Cfg_SpeedRefEUMax,Cfg_SpeedRefEUMin) MOV(Cfg_SpeedRefEUMin,Val_SpeedRefEUMax) MOV(Cfg_SpeedRefEUMax,Val_SpeedRefEUMin) ,LES(Cfg_OutDatalinkMin,Cfg_OutDatalinkEUMin) MOV(Cfg_OutDatalinkEUMin,Cfg_OutDatalinkMin) ,GRT(Cfg_OutDatalinkMin,Cfg_OutDatalinkEUMax) MOV(Cfg_OutDatalinkEUMax,Cfg_OutDatalinkMin) ,LES(Cfg_OutDatalinkMax,Cfg_OutDatalinkEUMin) MOV(Cfg_OutDatalinkEUMin,Cfg_OutDatalinkMax) ,GRT(Cfg_OutDatalinkMax,Cfg_OutDatalinkEUMax) MOV(Cfg_OutDatalinkEUMax,Cfg_OutDatalinkMax) ,LIM(7,Cfg_DecPlcs,-1) MOV(2,Cfg_DecPlcs) ,LIM(7,Cfg_InpDLDecPlcs,-1) MOV(2,Cfg_InpDLDecPlcs) ,LIM(7,Cfg_OutDLDecPlcs,-1) MOV(2,Cfg_OutDLDecPlcs) ];
